  MoveL 5679 to (450.81, 542.83, 100) mm, rotated rx -180 ry 0 rz 160 deg; joints [12.921, 56.747, 9.735, -144.774, 70.43, 166.693]
  Set speed (17.9 mm/s)
  Call Extruder(398.90582)
  MoveL 5680 to (450.02, 541.91, 100) mm, rotated rx 180 ry 0 rz 160 deg; joints [12.82, 56.625, 10.008, -144.909, 70.53, 166.82]
  Set speed (17.9 mm/s)
  Call Extruder(404.31502)
  MoveL 5681 to (448.94, 540.59, 100) mm, rotated rx -180 ry 0 rz 160 deg; joints [12.672, 56.455, 10.386, -145.103, 70.667, 166.997]
  Set speed (17.9 mm/s)
  Call Extruder(407.73007)
  MoveL 5682 to (448.28, 539.73, 100) mm, rotated rx 180 ry 0 rz 160 deg; joints [12.576, 56.35, 10.619, -145.229, 70.751, 167.108]
  Set speed (17.9 mm/s)
  Call Extruder(411.96935)
  MoveL 5683 to (447.47, 538.66, 100) mm, rotated rx -180 ry 0 rz 160 deg; joints [12.453, 56.223, 10.904, -145.387, 70.853, 167.245]
  Set speed (17.9 mm/s)
  Call Extruder(416.06322)
  MoveL 5684 to (446.71, 537.6, 100) mm, rotated rx 180 ry 0 rz 160 deg; joints [12.331, 56.102, 11.173, -145.543, 70.949, 167.375]
  Set speed (17.9 mm/s)
  Call Extruder(420.86880)
  MoveL 5685 to (445.85, 536.35, 100) mm, rotated rx 180 ry 0 rz 160 deg; joints [12.183, 55.965, 11.481, -145.728, 71.057, 167.526]
  Set speed (17.9 mm/s)
  Call Extruder(424.00300)
  MoveL 5686 to (445.3, 535.52, 100) mm, rotated rx 180 ry 0 rz 160 deg; joints [12.084, 55.877, 11.677, -145.851, 71.126, 167.624]
  Set speed (17.9 mm/s)
  Call Extruder(429.28945)
  MoveL 5687 to (444.4, 534.1, 100) mm, rotated rx 180 ry 0 rz 160 deg; joints [11.914, 55.733, 12, -146.061, 71.238, 167.787]
  Set speed (17.9 mm/s)
  Call Extruder(432.98156)
  MoveL 5688 to (443.8, 533.1, 100) mm, rotated rx 180 ry 0 rz 160 deg; joints [11.791, 55.636, 12.219, -146.211, 71.313, 167.899]
  Set speed (17.9 mm/s)
  Call Extruder(437.21112)
  MoveL 5689 to (443.13, 531.94, 100) mm, rotated rx -180 ry 0 rz 160 deg; joints [11.648, 55.527, 12.464, -146.384, 71.396, 168.025]
  Set speed (17.9 mm/s)
  Call Extruder(441.38194)
  MoveL 5690 to (442.49, 530.78, 100) mm, rotated rx -180 ry 0 rz 160 deg; joints [11.504, 55.423, 12.698, -146.557, 71.475, 168.149]
  Set speed (17.9 mm/s)
  Call Extruder(445.63460)
  MoveL 5691 to (441.87, 529.58, 100) mm, rotated rx 180 ry 0 rz 160 deg; joints [11.353, 55.32, 12.93, -146.736, 71.552, 168.273]
  Set speed (17.9 mm/s)
  Call Extruder(449.79410)
  MoveL 5692 to (441.29, 528.4, 100) mm, rotated rx -180 ry 0 rz 160 deg; joints [11.203, 55.223, 13.149, -146.913, 71.624, 168.392]
  Set speed (17.9 mm/s)
  Call Extruder(454.54369)
  MoveL 5693 to (440.65, 527.04, 100) mm, rotated rx -180 ry 0 rz 160 deg; joints [11.028, 55.116, 13.39, -147.118, 71.701, 168.526]
  Set speed (17.9 mm/s)
  Call Extruder(458.16789)
  MoveL 5694 to (440.18, 525.99, 100) mm, rotated rx 180 ry 0 rz 160 deg; joints [10.893, 55.036, 13.571, -147.276, 71.759, 168.627]
  Call Extruder(462.55520)
  MoveL 5695 to (439.64, 524.71, 100) mm, rotated rx -180 ry 0 rz 160 deg; joints [10.725, 54.945, 13.778, -147.469, 71.824, 168.747]
  Call Extruder(466.58097)
  MoveL 5696 to (439.17, 523.52, 100) mm, rotated rx -180 ry 0 rz 160 deg; joints [10.569, 54.863, 13.964, -147.648, 71.881, 168.856]
  Set speed (17.9 mm/s)
  Call Extruder(470.98501)
  MoveL 5697 to (438.69, 522.21, 100) mm, rotated rx -180 ry 0 rz 160 deg; joints [10.395, 54.778, 14.157, -147.847, 71.939, 168.972]
  Set speed (17.9 mm/s)
  Call Extruder(475.05223)
  MoveL 5698 to (438.25, 521, 100) mm, rotated rx -180 ry 0 rz 160 deg; joints [10.233, 54.701, 14.33, -148.031, 71.99, 169.078]
  Set speed (17.9 mm/s)
  Call Extruder(479.39790)
  MoveL 5699 to (437.83, 519.69, 100) mm, rotated rx 180 ry 0 rz 160 deg; joints [10.056, 54.624, 14.505, -148.23, 72.04, 169.189]
  Call Extruder(483.42476)
  MoveL 5700 to (437.45, 518.47, 100) mm, rotated rx 180 ry 0 rz 160 deg; joints [9.891, 54.555, 14.662, -148.416, 72.084, 169.29]
  Set speed (17.9 mm/s)
  Call Extruder(487.83422)
  MoveL 5701 to (437.07, 517.13, 100) mm, rotated rx -180 ry 0 rz 160 deg; joints [9.707, 54.484, 14.823, -148.621, 72.127, 169.398]
  Set speed (17.9 mm/s)
  Call Extruder(491.89983)
  MoveL 5702 to (436.74, 515.89, 100) mm, rotated rx 180 ry 0 rz 160 deg; joints [9.535, 54.421, 14.966, -148.812, 72.164, 169.496]
  Set speed (17.9 mm/s)
  Call Extruder(495.65111)
  MoveL 5703 to (436.47, 514.73, 100) mm, rotated rx -180 ry 0 rz 160 deg; joints [9.375, 54.367, 15.09, -148.989, 72.194, 169.584]
  Set speed (17.8 mm/s)
  Call Extruder(501.06220)
  MoveL 5704 to (436.1, 513.06, 100) mm, rotated rx 180 ry 0 rz 160 deg; joints [9.142, 54.293, 15.259, -149.245, 72.234, 169.709]
  Set speed (17.9 mm/s)
  Call Extruder(508.92492)
  MoveL 5705 to (435.64, 510.61, 100) mm, rotated rx -180 ry 0 rz 160 deg; joints [8.797, 54.196, 15.481, -149.622, 72.28, 169.884]
  Set speed (17.9 mm/s)
  Call Extruder(517.34016)
  MoveL 5706 to (435.26, 507.97, 100) mm, rotated rx 180 ry 0 rz 160 deg; joints [8.421, 54.106, 15.687, -150.03, 72.315, 170.064]
  Set speed (17.9 mm/s)
  Call Extruder(525.75236)
  MoveL 5707 to (435, 505.32, 100) mm, rotated rx 180 ry 0 rz 160 deg; joints [8.039, 54.031, 15.859, -150.44, 72.333, 170.234]
  Set speed (17.9 mm/s)
  Call Extruder(534.00913)
  MoveL 5708 to (434.83, 502.7, 100) mm, rotated rx -180 ry 0 rz 160 deg; joints [7.66, 53.971, 15.996, -150.844, 72.337, 170.393]
  Set speed (17.9 mm/s)
  Call Extruder(542.49356)
  MoveL 5709 to (434.77, 500.01, 100) mm, rotated rx 180 ry 0 rz 160 deg; joints [7.266, 53.923, 16.105, -151.261, 72.325, 170.547]
  Set speed (17.9 mm/s)
  Call Extruder(550.14962)
  MoveL 5710 to (434.82, 497.58, 100) mm, rotated rx 180 ry 0 rz 160 deg; joints [6.909, 53.894, 16.172, -151.637, 72.3, 170.679]
  Set speed (17.9 mm/s)
  Call Extruder(557.57595)
  MoveL 5711 to (434.95, 495.23, 100) mm, rotated rx 180 ry 0 rz 160 deg; joints [6.561, 53.877, 16.21, -152.001, 72.263, 170.799]
  Set speed (17.9 mm/s)
  Call Extruder(565.20370)
  MoveL 5712 to (435.17, 492.83, 100) mm, rotated rx 180 ry 0 rz 160 deg; joints [6.203, 53.871, 16.223, -152.373, 72.213, 170.916]
  Set speed (17.9 mm/s)
  Call Extruder(572.77473)
  MoveL 5713 to (435.48, 490.44, 100) mm, rotated rx -180 ry 0 rz 160 deg; joints [5.847, 53.878, 16.208, -152.741, 72.15, 171.025]
  Call Extruder(580.43460)
  MoveL 5714 to (435.88, 488.05, 100) mm, rotated rx 180 ry 0 rz 160 deg; joints [5.488, 53.897, 16.165, -153.11, 72.072, 171.128]
  Set speed (17.9 mm/s)
  Call Extruder(587.90471)
  MoveL 5715 to (436.36, 485.73, 100) mm, rotated rx -180 ry 0 rz 160 deg; joints [5.139, 53.927, 16.096, -153.466, 71.984, 171.221]
  Set speed (17.9 mm/s)
  Call Extruder(595.43174)
  MoveL 5716 to (436.92, 483.41, 100) mm, rotated rx 180 ry 0 rz 160 deg; joints [4.791, 53.969, 16, -153.821, 71.883, 171.308]
  Set speed (17.9 mm/s)
  Call Extruder(602.95230)
  MoveL 5717 to (437.57, 481.11, 100) mm, rotated rx 180 ry 0 rz 160 deg; joints [4.445, 54.023, 15.877, -154.171, 71.768, 171.389]
  Set speed (17.9 mm/s)
  Call Extruder(610.57330)
  MoveL 5718 to (438.32, 478.81, 100) mm, rotated rx -180 ry 0 rz 160 deg; joints [4.098, 54.089, 15.725, -154.52, 71.64, 171.463]
  Set speed (17.9 mm/s)
  Call Extruder(618.19372)
  MoveL 5719 to (439.14, 476.54, 100) mm, rotated rx -180 ry 0 rz 160 deg; joints [3.756, 54.167, 15.547, -154.862, 71.499, 171.531]
  Set speed (17.9 mm/s)
  Call Extruder(624.98487)
  MoveL 5720 to (439.95, 474.55, 100) mm, rotated rx 180 ry 0 rz 160 deg; joints [3.456, 54.246, 15.366, -155.161, 71.362, 171.585]
  Set speed (17.9 mm/s)
  Call Extruder(633.35469)
  MoveL 5721 to (441.03, 472.13, 100) mm, rotated rx 180 ry 0 rz 160 deg; joints [3.092, 54.357, 15.113, -155.521, 71.18, 171.645]
  Set speed (17.9 mm/s)
  Call Extruder(641.01629)
  MoveL 5722 to (442.11, 469.95, 100) mm, rotated rx 180 ry 0 rz 160 deg; joints [2.766, 54.471, 14.854, -155.842, 71, 171.692]
  Set speed (17.9 mm/s)
  Call Extruder(648.40572)
  MoveL 5723 to (443.23, 467.89, 100) mm, rotated rx -180 ry 0 rz 160 deg; joints [2.458, 54.591, 14.579, -156.142, 70.815, 171.731]
  Call Extruder(655.93186)
  MoveL 5724 to (444.44, 465.84, 100) mm, rotated rx 180 ry 0 rz 160 deg; joints [2.152, 54.725, 14.275, -156.439, 70.615, 171.764]
  Set speed (17.9 mm/s)
  Call Extruder(663.53574)
  MoveL 5725 to (445.74, 463.81, 100) mm, rotated rx -180 ry 0 rz 160 deg; joints [1.85, 54.872, 13.943, -156.73, 70.402, 171.792]
  Set speed (17.9 mm/s)
  Call Extruder(671.21430)
  MoveL 5726 to (447.13, 461.81, 100) mm, rotated rx 180 ry 0 rz 160 deg; joints [1.555, 55.031, 13.583, -157.012, 70.175, 171.813]
  Set speed (17.9 mm/s)
  Call Extruder(678.78294)
  MoveL 5727 to (448.57, 459.89, 100) mm, rotated rx 180 ry 0 rz 160 deg; joints [1.273, 55.199, 13.204, -157.279, 69.94, 171.826]
  Set speed (17.9 mm/s)
  Call Extruder(686.29697)
  MoveL 5728 to (450.07, 458.03, 100) mm, rotated rx 180 ry 0 rz 160 deg; joints [1.003, 55.376, 12.805, -157.533, 69.696, 171.834]
  Set speed (17.9 mm/s)
  Call Extruder(693.99931)
  MoveL 5729 to (451.68, 456.19, 100) mm, rotated rx 180 ry 0 rz 160 deg; joints [0.736, 55.568, 12.372, -157.781, 69.436, 171.835]
  Set speed (17.9 mm/s)
  Call Extruder(701.57500)
  MoveL 5730 to (453.33, 454.44, 100) mm, rotated rx -180 ry 0 rz 160 deg; joints [0.483, 55.767, 11.924, -158.012, 69.17, 171.829]
  Set speed (17.9 mm/s)
  Call Extruder(709.05583)
  MoveL 5731 to (455.02, 452.77, 100) mm, rotated rx -180 ry 0 rz 160 deg; joints [0.245, 55.974, 11.461, -158.228, 68.898, 171.817]
  Set speed (17.9 mm/s)
  Call Extruder(716.62216)
  MoveL 5732 to (456.79, 451.15, 100) mm, rotated rx 180 ry 0 rz 160 deg; joints [0.015, 56.193, 10.971, -158.433, 68.613, 171.798]
  Set speed (17.9 mm/s)
  Call Extruder(724.28486)
  MoveL 5733 to (458.64, 449.58, 100) mm, rotated rx -180 ry 0 rz 160 deg; joints [-0.206, 56.424, 10.454, -158.628, 68.316, 171.773]
  Set speed (17.9 mm/s)
  Call Extruder(731.69796)
  MoveL 5734 to (460.48, 448.12, 100) mm, rotated rx 180 ry 0 rz 160 deg; joints [-0.409, 56.657, 9.935, -158.803, 68.021, 171.741]
  Call Extruder(739.18151)
  MoveL 5735 to (462.39, 446.71, 100) mm, rotated rx -180 ry 0 rz 160 deg; joints [-0.603, 56.901, 9.393, -158.966, 67.715, 171.703]
  Set speed (17.9 mm/s)
  Call Extruder(746.80614)
  MoveL 5736 to (464.4, 445.36, 100) mm, rotated rx 180 ry 0 rz 160 deg; joints [-0.788, 57.159, 8.821, -159.117, 67.395, 171.657]
  Set speed (17.9 mm/s)
  Call Extruder(754.56977)
  MoveL 5737 to (466.48, 444.05, 100) mm, rotated rx -180 ry 0 rz 160 deg; joints [-0.964, 57.431, 8.221, -159.257, 67.062, 171.604]
  Call Extruder(762.12836)
  MoveL 5738 to (468.56, 442.86, 100) mm, rotated rx -180 ry 0 rz 160 deg; joints [-1.122, 57.703, 7.62, -159.378, 66.731, 171.545]
  Set speed (17.9 mm/s)
  Call Extruder(769.52658)
  MoveL 5739 to (470.63, 441.76, 100) mm, rotated rx -180 ry 0 rz 160 deg; joints [-1.266, 57.978, 7.015, -159.483, 66.401, 171.48]
  Call Extruder(777.24414)
  MoveL 5740 to (472.84, 440.7, 100) mm, rotated rx -180 ry 0 rz 160 deg; joints [-1.403, 58.272, 6.369, -159.577, 66.051, 171.405]
  Set speed (17.9 mm/s)
  Call Extruder(784.59819)
  MoveL 5741 to (474.98, 439.77, 100) mm, rotated rx 180 ry 0 rz 160 deg; joints [-1.522, 58.56, 5.738, -159.653, 65.712, 171.327]
  Set speed (17.9 mm/s)
  Call Extruder(792.28153)
  MoveL 5742 to (477.25, 438.88, 100) mm, rotated rx -180 ry 0 rz 160 deg; joints [-1.634, 58.869, 5.065, -159.716, 65.353, 171.238]
  Set speed (17.9 mm/s)
  Call Extruder(800.00638)
  MoveL 5743 to (479.56, 438.07, 100) mm, rotated rx -180 ry 0 rz 160 deg; joints [-1.733, 59.186, 4.374, -159.764, 64.987, 171.141]
  Set speed (17.9 mm/s)
  Call Extruder(807.42236)
  MoveL 5744 to (481.8, 437.37, 100) mm, rotated rx -180 ry 0 rz 160 deg; joints [-1.817, 59.497, 3.698, -159.796, 64.631, 171.04]
  Call Extruder(814.93635)
  MoveL 5745 to (484.1, 436.75, 100) mm, rotated rx 180 ry 0 rz 160 deg; joints [-1.89, 59.818, 3.002, -159.814, 64.268, 170.931]
  Set speed (17.9 mm/s)
  Call Extruder(822.70712)
  MoveL 5746 to (486.5, 436.19, 100) mm, rotated rx -180 ry 0 rz 160 deg; joints [-1.952, 60.156, 2.27, -159.816, 63.889, 170.81]
  Set speed (17.9 mm/s)
  Call Extruder(830.13943)
  MoveL 5747 to (488.82, 435.74, 100) mm, rotated rx 180 ry 0 rz 160 deg; joints [-2, 60.486, 1.559, -159.804, 63.523, 170.687]
  Set speed (17.9 mm/s)
  Call Extruder(837.63896)
  MoveL 5748 to (491.17, 435.38, 100) mm, rotated rx 180 ry 0 rz 160 deg; joints [-2.037, 60.823, 0.833, -159.778, 63.152, 170.555]
  Set speed (17.9 mm/s)
  Call Extruder(845.39030)
  MoveL 5749 to (493.61, 435.09, 100) mm, rotated rx 180 ry 0 rz 160 deg; joints [-2.063, 61.177, 0.074, -159.735, 62.767, 170.41]
  Call Extruder(852.91708)
  MoveL 5750 to (495.99, 434.9, 100) mm, rotated rx 180 ry 0 rz 160 deg; joints [-2.076, 61.525, -0.672, -159.678, 62.392, 170.261]
  Set speed (17.9 mm/s)
  Call Extruder(860.57094)
  MoveL 5751 to (498.41, 434.8, 100) mm, rotated rx 180 ry 0 rz 160 deg; joints [-2.078, 61.883, -1.437, -159.605, 62.01, 170.102]
  Set speed (17.9 mm/s)
  Call Extruder(868.06031)
  MoveL 5752 to (500.79, 434.78, 100) mm, rotated rx 180 ry 0 rz 160 deg; joints [-2.069, 62.237, -2.193, -159.52, 61.636, 169.939]
  Call Extruder(875.70122)
  MoveL 5753 to (503.21, 434.86, 100) mm, rotated rx -180 ry 0 rz 160 deg; joints [-2.049, 62.602, -2.969, -159.419, 61.254, 169.763]
  Set speed (17.9 mm/s)
  Call Extruder(883.20616)
  MoveL 5754 to (505.59, 435.02, 100) mm, rotated rx 180 ry 0 rz 160 deg; joints [-2.018, 62.963, -3.736, -159.305, 60.88, 169.583]
  Set speed (17.9 mm/s)
  Call Extruder(890.83877)
  MoveL 5755 to (508, 435.27, 100) mm, rotated rx 180 ry 0 rz 160 deg; joints [-1.976, 63.333, -4.52, -159.175, 60.501, 169.392]
  Call Extruder(898.35749)
  MoveL 5756 to (510.35, 435.61, 100) mm, rotated rx 180 ry 0 rz 160 deg; joints [-1.924, 63.7, -5.294, -159.033, 60.129, 169.195]
  Set speed (17.9 mm/s)
  Call Extruder(905.98584)
  MoveL 5757 to (512.74, 436.03, 100) mm, rotated rx -180 ry 0 rz 160 deg; joints [-1.861, 64.074, -6.083, -158.876, 59.754, 168.987]
  Call Extruder(913.34804)
  MoveL 5758 to (515.02, 436.53, 100) mm, rotated rx 180 ry 0 rz 160 deg; joints [-1.79, 64.436, -6.845, -158.711, 59.395, 168.779]
  Call Extruder(920.98532)
  MoveL 5759 to (517.37, 437.13, 100) mm, rotated rx 180 ry 0 rz 160 deg; joints [-1.707, 64.813, -7.637, -158.526, 59.025, 168.555]
  Set speed (17.9 mm/s)
  Call Extruder(928.62246)
  MoveL 5760 to (519.69, 437.82, 100) mm, rotated rx 180 ry 0 rz 160 deg; joints [-1.615, 65.19, -8.427, -158.328, 58.659, 168.322]
  Set speed (17.9 mm/s)
  Call Extruder(936.05332)
  MoveL 5761 to (521.92, 438.57, 100) mm, rotated rx -180 ry 0 rz 160 deg; joints [-1.516, 65.557, -9.195, -158.124, 58.307, 168.088]
  Call Extruder(943.74007)
  MoveL 5762 to (524.21, 439.43, 100) mm, rotated rx -180 ry 0 rz 160 deg; joints [-1.404, 65.936, -9.986, -157.899, 57.948, 167.839]
  Set speed (17.9 mm/s)
  Call Extruder(951.26725)
  MoveL 5763 to (526.4, 440.36, 100) mm, rotated rx 180 ry 0 rz 160 deg; joints [-1.286, 66.306, -10.757, -157.667, 57.602, 167.587]
  Call Extruder(958.89094)
  MoveL 5764 to (528.6, 441.38, 100) mm, rotated rx 180 ry 0 rz 160 deg; joints [-1.158, 66.68, -11.534, -157.42, 57.257, 167.324]
  Call Extruder(966.54138)
  MoveL 5765 to (530.76, 442.49, 100) mm, rotated rx -180 ry 0 rz 160 deg; joints [-1.021, 67.053, -12.308, -157.161, 56.917, 167.053]
  Call Extruder(974.10055)
  MoveL 5766 to (532.85, 443.66, 100) mm, rotated rx 180 ry 0 rz 160 deg; joints [-0.878, 67.419, -13.067, -156.894, 56.589, 166.779]
  Set speed (17.9 mm/s)
  Call Extruder(981.59160)
  MoveL 5767 to (534.88, 444.89, 100) mm, rotated rx 180 ry 0 rz 160 deg; joints [-0.728, 67.778, -13.811, -156.618, 56.27, 166.5]
  Set speed (17.9 mm/s)
  Call Extruder(989.24433)
  MoveL 5768 to (536.91, 446.23, 100) mm, rotated rx 180 ry 0 rz 160 deg; joints [-0.567, 68.142, -14.562, -156.326, 55.953, 166.209]
  Set speed (17.9 mm/s)
  Call Extruder(996.72405)
  MoveL 5769 to (538.84, 447.6, 100) mm, rotated rx -180 ry 0 rz 160 deg; joints [-0.404, 68.493, -15.287, -156.032, 55.651, 165.918]
  Set speed (17.9 mm/s)
  Call Extruder(1004.30520)
  MoveL 5770 to (540.75, 449.07, 100) mm, rotated rx -180 ry 0 rz 160 deg; joints [-0.23, 68.845, -16.01, -155.723, 55.354, 165.618]
  Set speed (17.9 mm/s)
  Call Extruder(1011.81497)
  MoveL 5771 to (542.58, 450.59, 100) mm, rotated rx 180 ry 0 rz 160 deg; joints [-0.052, 69.188, -16.715, -155.409, 55.069, 165.316]
  Set speed (17.9 mm/s)
  Call Extruder(1019.44561)
  MoveL 5772 to (544.38, 452.21, 100) mm, rotated rx -180 ry 0 rz 160 deg; joints [0.135, 69.531, -17.419, -155.082, 54.789, 165.005]
  Set speed (17.9 mm/s)
  Call Extruder(1026.97139)
  MoveL 5773 to (546.1, 453.86, 100) mm, rotated rx 180 ry 0 rz 160 deg; joints [0.326, 69.862, -18.098, -154.751, 54.524, 164.693]
  Set speed (17.9 mm/s)
  Call Extruder(1031.19963)
  MoveL 5774 to (547.04, 454.82, 100) mm, rotated rx -180 ry 0 rz 160 deg; joints [0.436, 70.046, -18.474, -154.562, 54.379, 164.516]
  Set speed (17.9 mm/s)
  Call Extruder(1035.37002)
  MoveL 5775 to (547.94, 455.78, 100) mm, rotated rx -180 ry 0 rz 160 deg; joints [0.546, 70.225, -18.84, -154.374, 54.24, 164.341]
  Set speed (17.9 mm/s)
  Call Extruder(1038.63837)
  MoveL 5776 to (548.64, 456.55, 100) mm, rotated rx -180 ry 0 rz 160 deg; joints [0.634, 70.364, -19.124, -154.224, 54.133, 164.202]
  Set speed (17.9 mm/s)
  Call Extruder(1044.28026)
  MoveL 5777 to (549.82, 457.9, 100) mm, rotated rx -180 ry 0 rz 160 deg; joints [0.787, 70.599, -19.605, -153.964, 53.954, 163.962]
  Set speed (17.9 mm/s)
  Call Extruder(1047.97187)
  MoveL 5778 to (550.56, 458.8, 100) mm, rotated rx -180 ry 0 rz 160 deg; joints [0.889, 70.751, -19.915, -153.792, 53.841, 163.805]
  Set speed (17.9 mm/s)
  Call Extruder(1052.40017)
  MoveL 5779 to (551.44, 459.9, 100) mm, rotated rx 180 ry 0 rz 160 deg; joints [1.013, 70.93, -20.281, -153.584, 53.708, 163.615]
  Call Extruder(1056.39533)
  MoveL 5780 to (552.21, 460.91, 100) mm, rotated rx 180 ry 0 rz 160 deg; joints [1.127, 71.089, -20.604, -153.395, 53.593, 163.444]
  Set speed (17.9 mm/s)
  Call Extruder(1060.64284)
  MoveL 5781 to (553, 461.99, 100) mm, rotated rx -180 ry 0 rz 160 deg; joints [1.249, 71.255, -20.943, -153.192, 53.474, 163.261]
  Set speed (17.9 mm/s)
  Call Extruder(1064.81823)
  MoveL 5782 to (553.76, 463.08, 100) mm, rotated rx 180 ry 0 rz 160 deg; joints [1.371, 71.416, -21.269, -152.991, 53.361, 163.081]
  Set speed (17.9 mm/s)
  Call Extruder(1069.00747)
  MoveL 5783 to (554.5, 464.18, 100) mm, rotated rx 180 ry 0 rz 160 deg; joints [1.494, 71.573, -21.59, -152.789, 53.252, 162.9]
  Set speed (17.9 mm/s)
  Call Extruder(1073.69401)
  MoveL 5784 to (555.31, 465.43, 100) mm, rotated rx 180 ry 0 rz 160 deg; joints [1.633, 71.747, -21.942, -152.561, 53.134, 162.698]
  Set speed (17.9 mm/s)
  Call Extruder(1077.43188)
  MoveL 5785 to (555.93, 466.44, 100) mm, rotated rx 180 ry 0 rz 160 deg; joints [1.746, 71.881, -22.216, -152.378, 53.045, 162.537]
  Call Extruder(1081.67784)
  MoveL 5786 to (556.61, 467.6, 100) mm, rotated rx -180 ry 0 rz 160 deg; joints [1.875, 72.031, -22.521, -152.17, 52.947, 162.354]
  Set speed (17.9 mm/s)
  Call Extruder(1087.53287)
  MoveL 5787 to (557.51, 469.23, 100) mm, rotated rx -180 ry 0 rz 160 deg; joints [2.055, 72.233, -22.929, -151.882, 52.819, 162.103]
  Set speed (17.9 mm/s)
  Call Extruder(1090.17409)
  MoveL 5788 to (557.9, 469.97, 100) mm, rotated rx -180 ry 0 rz 160 deg; joints [2.137, 72.321, -23.109, -151.751, 52.764, 161.99]
  Set speed (17.9 mm/s)
  Call Extruder(1094.24936)
  MoveL 5789 to (558.48, 471.12, 100) mm, rotated rx -180 ry 0 rz 160 deg; joints [2.264, 72.454, -23.379, -151.549, 52.683, 161.816]
  Set speed (17.9 mm/s)
  Call Extruder(1098.95352)
  MoveL 5790 to (559.12, 472.47, 100) mm, rotated rx 180 ry 0 rz 160 deg; joints [2.413, 72.604, -23.682, -151.316, 52.595, 161.616]
  Set speed (17.9 mm/s)
  Call Extruder(1102.65916)
  MoveL 5791 to (559.61, 473.54, 100) mm, rotated rx 180 ry 0 rz 160 deg; joints [2.531, 72.718, -23.914, -151.132, 52.529, 161.459]
  Set speed (17.9 mm/s)
  Call Extruder(1107.37343)
  MoveL 5792 to (560.2, 474.91, 100) mm, rotated rx 180 ry 0 rz 160 deg; joints [2.682, 72.858, -24.196, -150.898, 52.452, 161.262]
  Set speed (17.9 mm/s)
  Call Extruder(1111.28917)
  MoveL 5793 to (560.67, 476.06, 100) mm, rotated rx -180 ry 0 rz 160 deg; joints [2.808, 72.972, -24.428, -150.703, 52.391, 161.098]
  Call Extruder(1115.41542)
  MoveL 5794 to (561.13, 477.28, 100) mm, rotated rx 180 ry 0 rz 160 deg; joints [2.943, 73.086, -24.658, -150.499, 52.333, 160.928]
  Set speed (17.9 mm/s)
  Call Extruder(1119.53817)
  MoveL 5795 to (561.58, 478.5, 100) mm, rotated rx -180 ry 0 rz 160 deg; joints [3.077, 73.199, -24.885, -150.294, 52.278, 160.758]
  Set speed (17.9 mm/s)
  Call Extruder(1123.83675)
  MoveL 5796 to (562.01, 479.8, 100) mm, rotated rx -180 ry 0 rz 160 deg; joints [3.219, 73.308, -25.107, -150.082, 52.227, 160.584]
  Call Extruder(1128.03874)
  MoveL 5797 to (562.41, 481.06, 100) mm, rotated rx 180 ry 0 rz 160 deg; joints [3.358, 73.414, -25.32, -149.875, 52.18, 160.414]
  Set speed (17.9 mm/s)
  Call Extruder(1132.22902)
  MoveL 5798 to (562.78, 482.34, 100) mm, rotated rx -180 ry 0 rz 160 deg; joints [3.497, 73.512, -25.518, -149.669, 52.141, 160.248]
  Set speed (17.9 mm/s)
  Call Extruder(1136.26465)
  MoveL 5799 to (563.12, 483.57, 100) mm, rotated rx 180 ry 0 rz 160 deg; joints [3.632, 73.605, -25.705, -149.471, 52.106, 160.089]
  Call Extruder(1140.67454)
  MoveL 5800 to (563.45, 484.93, 100) mm, rotated rx -180 ry 0 rz 160 deg; joints [3.781, 73.698, -25.895, -149.256, 52.074, 159.918]
  Call Extruder(1144.77390)
  MoveL 5801 to (563.74, 486.19, 100) mm, rotated rx 180 ry 0 rz 160 deg; joints [3.919, 73.784, -26.066, -149.057, 52.048, 159.761]
  Set speed (17.9 mm/s)
  Call Extruder(1153.44625)
  MoveL 5802 to (564.27, 488.89, 100) mm, rotated rx 180 ry 0 rz 160 deg; joints [4.215, 73.945, -26.391, -148.639, 52.01, 159.437]
  Set speed (17.9 mm/s)
  Call Extruder(1161.67703)
  MoveL 5803 to (564.66, 491.47, 100) mm, rotated rx 180 ry 0 rz 160 deg; joints [4.498, 74.078, -26.66, -148.248, 51.995, 159.14]
  Call Extruder(1170.18168)
  MoveL 5804 to (564.96, 494.15, 100) mm, rotated rx -180 ry 0 rz 160 deg; joints [4.792, 74.196, -26.897, -147.85, 51.999, 158.845]
  Call Extruder(1178.50578)
  MoveL 5805 to (565.14, 496.79, 100) mm, rotated rx 180 ry 0 rz 160 deg; joints [5.082, 74.29, -27.086, -147.468, 52.024, 158.57]
  Set speed (17.9 mm/s)
  Call Extruder(1186.85602)
  MoveL 5806 to (565.22, 499.43, 100) mm, rotated rx 180 ry 0 rz 160 deg; joints [5.373, 74.362, -27.232, -147.093, 52.069, 158.308]
  Set speed (17.9 mm/s)
  Call Extruder(1195.19846)
  MoveL 5807 to (565.19, 502.08, 100) mm, rotated rx -180 ry 0 rz 160 deg; joints [5.665, 74.414, -27.336, -146.727, 52.134, 158.061]
  Set speed (17.9 mm/s)
  Call Extruder(1203.73141)
  MoveL 5808 to (565.05, 504.78, 100) mm, rotated rx 180 ry 0 rz 160 deg; joints [5.965, 74.445, -27.399, -146.362, 52.22, 157.824]
  Set speed (17.9 mm/s)
  Call Extruder(1212.05652)
  MoveL 5809 to (564.8, 507.41, 100) mm, rotated rx -180 ry 0 rz 160 deg; joints [6.258, 74.453, -27.414, -146.016, 52.325, 157.609]
  Set speed (17.9 mm/s)
  Call Extruder(1220.63729)
  MoveL 5810 to (564.43, 510.11, 100) mm, rotated rx -180 ry 0 rz 160 deg; joints [6.559, 74.438, -27.385, -145.671, 52.453, 157.404]
  Call Extruder(1229.19039)
  MoveL 5811 to (563.96, 512.78, 100) mm, rotated rx 180 ry 0 rz 160 deg; joints [6.859, 74.401, -27.31, -145.338, 52.599, 157.219]
  Call Extruder(1237.40699)
  MoveL 5812 to (563.39, 515.33, 100) mm, rotated rx 180 ry 0 rz 160 deg; joints [7.147, 74.344, -27.195, -145.03, 52.759, 157.058]
  Set speed (17.9 mm/s)
  Call Extruder(1245.34913)
  MoveL 5813 to (562.76, 517.76, 100) mm, rotated rx -180 ry 0 rz 160 deg; joints [7.424, 74.269, -27.045, -144.743, 52.928, 156.92]
  Set speed (17.9 mm/s)
  Call Extruder(1250.95485)
  MoveL 5814 to (562.25, 519.46, 100) mm, rotated rx 180 ry 0 rz 160 deg; joints [7.618, 74.204, -26.914, -144.548, 53.059, 156.833]
  Set speed (17.9 mm/s)
  Call Extruder(1254.21125)
  MoveL 5815 to (561.94, 520.45, 100) mm, rotated rx 180 ry 0 rz 160 deg; joints [7.731, 74.164, -26.833, -144.436, 53.136, 156.785]
  Call Extruder(1258.88399)
  MoveL 5816 to (561.45, 521.84, 100) mm, rotated rx 180 ry 0 rz 160 deg; joints [7.892, 74.097, -26.698, -144.281, 53.255, 156.723]
  Set speed (17.9 mm/s)
  Call Extruder(1262.79210)
  MoveL 5817 to (561.03, 523.01, 100) mm, rotated rx -180 ry 0 rz 160 deg; joints [8.027, 74.039, -26.581, -144.152, 53.356, 156.674]
  Set speed (17.9 mm/s)
  Call Extruder(1267.25552)
  MoveL 5818 to (560.51, 524.33, 100) mm, rotated rx 180 ry 0 rz 160 deg; joints [8.18, 73.965, -26.431, -144.01, 53.478, 156.625]
  Call Extruder(1270.87292)
  MoveL 5819 to (560.08, 525.39, 100) mm, rotated rx 180 ry 0 rz 160 deg; joints [8.304, 73.902, -26.306, -143.896, 53.578, 156.587]
  Call Extruder(1275.66647)
  MoveL 5820 to (559.47, 526.78, 100) mm, rotated rx 180 ry 0 rz 160 deg; joints [8.467, 73.812, -26.123, -143.75, 53.718, 156.544]
  Set speed (17.9 mm/s)
  Call Extruder(1279.88602)
  MoveL 5821 to (558.91, 527.99, 100) mm, rotated rx -180 ry 0 rz 160 deg; joints [8.61, 73.729, -25.955, -143.624, 53.843, 156.51]
  Set speed (17.9 mm/s)
  Call Extruder(1283.61536)
  MoveL 5822 to (558.39, 529.06, 100) mm, rotated rx -180 ry 0 rz 160 deg; joints [8.736, 73.65, -25.796, -143.516, 53.957, 156.485]
  Set speed (17.9 mm/s)
  Call Extruder(1287.99352)
  MoveL 5823 to (557.76, 530.29, 100) mm, rotated rx -180 ry 0 rz 160 deg; joints [8.884, 73.552, -25.6, -143.392, 54.096, 156.46]
  Set speed (17.9 mm/s)
  Call Extruder(1292.53711)
  MoveL 5824 to (557.07, 531.56, 100) mm, rotated rx 180 ry 0 rz 160 deg; joints [9.035, 73.446, -25.385, -143.267, 54.244, 156.439]
  Call Extruder(1296.24969)
  MoveL 5825 to (556.5, 532.59, 100) mm, rotated rx -180 ry 0 rz 160 deg; joints [9.159, 73.355, -25.202, -143.167, 54.367, 156.426]
  Set speed (17.9 mm/s)
  Call Extruder(1300.41758)
  MoveL 5826 to (555.83, 533.73, 100) mm, rotated rx -180 ry 0 rz 160 deg; joints [9.297, 73.25, -24.988, -143.058, 54.508, 156.415]
  Set speed (17.9 mm/s)
  Call Extruder(1304.83583)
  MoveL 5827 to (555.09, 534.92, 100) mm, rotated rx -180 ry 0 rz 160 deg; joints [9.442, 73.133, -24.752, -142.946, 54.662, 156.409]
  Set speed (17.9 mm/s)
  Call Extruder(1308.83293)
  MoveL 5828 to (554.4, 535.99, 100) mm, rotated rx -180 ry 0 rz 160 deg; joints [9.572, 73.022, -24.529, -142.848, 54.804, 156.407]
  Set speed (17.9 mm/s)
  Call Extruder(1313.12375)
  MoveL 5829 to (553.63, 537.11, 100) mm, rotated rx 180 ry 0 rz 160 deg; joints [9.711, 72.899, -24.28, -142.746, 54.96, 156.411]
  Set speed (17.9 mm/s)
  Call Extruder(1317.41236)
  MoveL 5830 to (552.85, 538.22, 100) mm, rotated rx 180 ry 0 rz 160 deg; joints [9.849, 72.773, -24.024, -142.646, 55.118, 156.418]
  Set speed (17.9 mm/s)
  Call Extruder(1322.92340)
  MoveL 5831 to (551.81, 539.63, 100) mm, rotated rx 180 ry 0 rz 160 deg; joints [10.025, 72.604, -23.682, -142.523, 55.326, 156.434]
  Set speed (17.9 mm/s)
  Call Extruder(1325.83347)
  MoveL 5832 to (551.24, 540.35, 100) mm, rotated rx 180 ry 0 rz 160 deg; joints [10.117, 72.512, -23.496, -142.461, 55.437, 156.446]
  Set speed (17.9 mm/s)
  Call Extruder(1329.94289)
  MoveL 5833 to (550.43, 541.37, 100) mm, rotated rx -180 ry 0 rz 160 deg; joints [10.246, 72.379, -23.226, -142.375, 55.597, 156.466]
  Set speed (17.9 mm/s)
  Call Extruder(1335.20101)
  MoveL 5834 to (549.35, 542.65, 100) mm, rotated rx -180 ry 0 rz 160 deg; joints [10.41, 72.204, -22.871, -142.268, 55.805, 156.497]
  Set speed (17.9 mm/s)
  Call Extruder(1338.74944)
  MoveL 5835 to (548.61, 543.49, 100) mm, rotated rx 180 ry 0 rz 160 deg; joints [10.519, 72.082, -22.623, -142.199, 55.948, 156.522]
  Set speed (17.9 mm/s)
  Call Extruder(1342.97071)
  MoveL 5836 to (547.7, 544.48, 100) mm, rotated rx 180 ry 0 rz 160 deg; joints [10.648, 71.933, -22.322, -142.12, 56.12, 156.556]
  Set speed (17.9 mm/s)
  Call Extruder(1347.16725)
  MoveL 5837 to (546.79, 545.44, 100) mm, rotated rx -180 ry 0 rz 160 deg; joints [10.774, 71.783, -22.017, -142.044, 56.292, 156.592]
  Set speed (17.9 mm/s)
  Call Extruder(1350.92435)
  MoveL 5838 to (545.95, 546.29, 100) mm, rotated rx 180 ry 0 rz 160 deg; joints [10.887, 71.645, -21.737, -141.978, 56.449, 156.629]
  Set speed (17.9 mm/s)
  Call Extruder(1355.12158)
  MoveL 5839 to (545, 547.22, 100) mm, rotated rx -180 ry 0 rz 160 deg; joints [11.011, 71.489, -21.418, -141.907, 56.626, 156.673]
  Set speed (17.9 mm/s)
  Call Extruder(1359.46484)
  MoveL 5840 to (543.99, 548.16, 100) mm, rotated rx -180 ry 0 rz 160 deg; joints [11.138, 71.323, -21.08, -141.837, 56.811, 156.724]
  Set speed (17.9 mm/s)
  Call Extruder(1363.56091)
  MoveL 5841 to (543.02, 549.02, 100) mm, rotated rx -180 ry 0 rz 160 deg; joints [11.256, 71.164, -20.756, -141.774, 56.988, 156.774]
  Call Extruder(1367.80541)
  MoveL 5842 to (542, 549.9, 100) mm, rotated rx 180 ry 0 rz 160 deg; joints [11.377, 70.996, -20.415, -141.711, 57.172, 156.83]
  Set speed (17.9 mm/s)
  Call Extruder(1371.93527)
  MoveL 5843 to (540.99, 550.73, 100) mm, rotated rx 180 ry 0 rz 160 deg; joints [11.494, 70.83, -20.076, -141.653, 57.353, 156.889]
  Call Extruder(1376.11842)
  MoveL 5844 to (539.95, 551.56, 100) mm, rotated rx -180 ry 0 rz 160 deg; joints [11.61, 70.659, -19.728, -141.596, 57.538, 156.951]
  Set speed (17.9 mm/s)
  Call Extruder(1380.34094)
  MoveL 5845 to (538.88, 552.37, 100) mm, rotated rx 180 ry 0 rz 160 deg; joints [11.726, 70.484, -19.371, -141.541, 57.726, 157.018]
  Call Extruder(1384.78388)
  MoveL 5846 to (537.74, 553.2, 100) mm, rotated rx -180 ry 0 rz 160 deg; joints [11.846, 70.298, -18.989, -141.487, 57.925, 157.092]
  Set speed (17.9 mm/s)
  Call Extruder(1389.23338)
  MoveL 5847 to (536.58, 554, 100) mm, rotated rx 180 ry 0 rz 160 deg; joints [11.964, 70.108, -18.6, -141.436, 58.127, 157.17]
  Set speed (17.9 mm/s)
  Call Extruder(1392.85535)
  MoveL 5848 to (535.62, 554.64, 100) mm, rotated rx -180 ry 0 rz 160 deg; joints [12.059, 69.951, -18.281, -141.396, 58.291, 157.235]
  Set speed (17.9 mm/s)
  Call Extruder(1397.17836)
  MoveL 5849 to (534.47, 555.37, 100) mm, rotated rx 180 ry 0 rz 160 deg; joints [12.17, 69.763, -17.894, -141.352, 58.489, 157.317]
  Set speed (17.9 mm/s)
  Call Extruder(1401.83512)
  MoveL 5850 to (533.21, 556.14, 100) mm, rotated rx 180 ry 0 rz 160 deg; joints [12.288, 69.557, -17.473, -141.307, 58.702, 157.409]
  Set speed (17.9 mm/s)
  Call Extruder(1405.59771)
  MoveL 5851 to (532.17, 556.74, 100) mm, rotated rx -180 ry 0 rz 160 deg; joints [12.382, 69.389, -17.127, -141.273, 58.876, 157.486]
  Set speed (17.9 mm/s)
  Call Extruder(1409.23758)
  MoveL 5852 to (531.16, 557.3, 100) mm, rotated rx 180 ry 0 rz 160 deg; joints [12.471, 69.225, -16.791, -141.242, 59.045, 157.562]
  Set speed (17.9 mm/s)
  Call Extruder(1414.04469)
  MoveL 5853 to (529.82, 558.01, 100) mm, rotated rx 180 ry 0 rz 160 deg; joints [12.586, 69.006, -16.342, -141.204, 59.269, 157.667]
  Call Extruder(1418.67857)
  MoveL 5854 to (528.5, 558.66, 100) mm, rotated rx -180 ry 0 rz 160 deg; joints [12.694, 68.793, -15.904, -141.171, 59.485, 157.772]
  Set speed (17.9 mm/s)
  Call Extruder(1422.53414)
  MoveL 5855 to (527.4, 559.19, 100) mm, rotated rx 180 ry 0 rz 160 deg; joints [12.783, 68.615, -15.536, -141.146, 59.666, 157.861]
  Set speed (17.9 mm/s)
  Call Extruder(1426.70274)
  MoveL 5856 to (526.19, 559.73, 100) mm, rotated rx -180 ry 0 rz 160 deg; joints [12.876, 68.42, -15.135, -141.122, 59.861, 157.961]
  Set speed (17.9 mm/s)
  Call Extruder(1430.81868)
  MoveL 5857 to (524.99, 560.24, 100) mm, rotated rx -180 ry 0 rz 160 deg; joints [12.966, 68.227, -14.738, -141.099, 60.054, 158.06]
  Set speed (17.9 mm/s)
  Call Extruder(1435.12111)
  MoveL 5858 to (523.73, 560.75, 100) mm, rotated rx 180 ry 0 rz 160 deg; joints [13.058, 68.024, -14.318, -141.079, 60.257, 158.168]
  Set speed (17.9 mm/s)
  Call Extruder(1439.34950)
  MoveL 5859 to (522.48, 561.23, 100) mm, rotated rx -180 ry 0 rz 160 deg; joints [13.146, 67.823, -13.904, -141.06, 60.456, 158.276]
  Set speed (17.9 mm/s)
  Call Extruder(1443.96614)
  MoveL 5860 to (521.1, 561.71, 100) mm, rotated rx 180 ry 0 rz 160 deg; joints [13.239, 67.602, -13.447, -141.045, 60.674, 158.398]
  Call Extruder(1447.75239)
  MoveL 5861 to (519.96, 562.09, 100) mm, rotated rx 180 ry 0 rz 160 deg; joints [13.315, 67.421, -13.072, -141.033, 60.852, 158.498]
  Set speed (17.9 mm/s)
  Call Extruder(1456.11391)
  MoveL 5862 to (517.42, 562.85, 100) mm, rotated rx -180 ry 0 rz 160 deg; joints [13.473, 67.016, -12.233, -141.016, 61.247, 158.729]
  Set speed (17.9 mm/s)
  Call Extruder(1459.84226)
  MoveL 5863 to (516.28, 563.15, 100) mm, rotated rx 180 ry 0 rz 160 deg; joints [13.539, 66.834, -11.856, -141.012, 61.423, 158.835]
  Set speed (17.9 mm/s)
  Call Extruder(1464.46214)
  MoveL 5864 to (514.86, 563.51, 100) mm, rotated rx -180 ry 0 rz 160 deg; joints [13.62, 66.61, -11.389, -141.009, 61.641, 158.967]
  Set speed (17.9 mm/s)
  Call Extruder(1473.02091)
  MoveL 5865 to (512.21, 564.07, 100) mm, rotated rx -180 ry 0 rz 160 deg; joints [13.762, 66.19, -10.516, -141.012, 62.044, 159.22]
  Call Extruder(1481.48428)
  MoveL 5866 to (509.56, 564.52, 100) mm, rotated rx 180 ry 0 rz 160 deg; joints [13.891, 65.774, -9.647, -141.025, 62.441, 159.478]
  Call Extruder(1489.72627)
  MoveL 5867 to (506.97, 564.85, 100) mm, rotated rx 180 ry 0 rz 160 deg; joints [14.006, 65.367, -8.797, -141.048, 62.825, 159.736]
  Set speed (17.9 mm/s)
  Call Extruder(1498.27519)
  MoveL 5868 to (504.26, 565.08, 100) mm, rotated rx -180 ry 0 rz 160 deg; joints [14.114, 64.945, -7.913, -141.082, 63.222, 160.01]
  Call Extruder(1506.73394)
  MoveL 5869 to (501.58, 565.2, 100) mm, rotated rx 180 ry 0 rz 160 deg; joints [14.209, 64.527, -7.037, -141.126, 63.611, 160.287]
  Set speed (17.9 mm/s)
  Call Extruder(1514.95462)
  MoveL 5870 to (498.98, 565.21, 100) mm, rotated rx 180 ry 0 rz 160 deg; joints [14.289, 64.123, -6.186, -141.179, 63.986, 160.562]
  Set speed (10.0 mm/s)
  MoveL 5871 to (498.98, 565.21, 104) mm, rotated rx 180 ry 0 rz 160 deg; joints [14.289, 63.491, -5.899, -141.073, 63.717, 160.321]
  Set speed (120.0 mm/s)
  MoveL 5872 to (498.98, 564.59, 104) mm, rotated rx -180 ry 0 rz 160 deg; joints [14.214, 63.467, -5.849, -141.16, 63.712, 160.374]
  Set speed (17.6 mm/s)
  Call Extruder(1523.55152)
  MoveL 5873 to (496.3, 564.49, 104) mm, rotated rx 180 ry 0 rz 160 deg; joints [14.285, 63.05, -4.975, -141.226, 64.092, 160.66]
  Set speed (17.6 mm/s)
  Call Extruder(1532.03521)
  MoveL 5874 to (493.65, 564.29, 104) mm, rotated rx 180 ry 0 rz 160 deg; joints [14.341, 62.641, -4.116, -141.302, 64.462, 160.947]
  Call Extruder(1540.42814)
  MoveL 5875 to (491.05, 563.98, 104) mm, rotated rx 180 ry 0 rz 160 deg; joints [14.385, 62.239, -3.269, -141.389, 64.823, 161.235]
  Set speed (17.6 mm/s)
  Call Extruder(1548.78688)
  MoveL 5876 to (488.47, 563.56, 104) mm, rotated rx 180 ry 0 rz 160 deg; joints [14.415, 61.841, -2.43, -141.486, 65.178, 161.525]
  Set speed (17.6 mm/s)
  Call Extruder(1557.21308)
  MoveL 5877 to (485.89, 563.04, 104) mm, rotated rx 180 ry 0 rz 160 deg; joints [14.432, 61.444, -1.59, -141.594, 65.53, 161.821]
  Set speed (17.6 mm/s)
  Call Extruder(1561.62651)
  MoveL 5878 to (484.55, 562.72, 104) mm, rotated rx -180 ry 0 rz 160 deg; joints [14.435, 61.238, -1.153, -141.655, 65.712, 161.977]
  Set speed (17.6 mm/s)
  Call Extruder(1565.84704)
  MoveL 5879 to (483.27, 562.4, 104) mm, rotated rx 180 ry 0 rz 160 deg; joints [14.436, 61.042, -0.738, -141.716, 65.884, 162.126]
  Set speed (17.6 mm/s)
  Call Extruder(1574.11726)
  MoveL 5880 to (480.8, 561.68, 104) mm, rotated rx 180 ry 0 rz 160 deg; joints [14.426, 60.661, 0.071, -141.844, 66.218, 162.42]
  Call Extruder(0.00000)
  Set speed (17.6 mm/s)
  Call Extruder(4.38070)
  MoveL 5881 to (479.5, 561.25, 104) mm, rotated rx -180 ry 0 rz 160 deg; joints [14.414, 60.462, 0.496, -141.917, 66.391, 162.577]
  Call Extruder(8.59213)
  MoveL 5882 to (478.25, 560.83, 104) mm, rotated rx -180 ry 0 rz 160 deg; joints [14.402, 60.271, 0.901, -141.988, 66.557, 162.727]
  Set speed (17.6 mm/s)
  Call Extruder(12.89777)
  MoveL 5883 to (477, 560.36, 104) mm, rotated rx 180 ry 0 rz 160 deg; joints [14.383, 60.078, 1.313, -142.066, 66.724, 162.881]
  Call Extruder(17.56272)
  MoveL 5884 to (475.64, 559.83, 104) mm, rotated rx 180 ry 0 rz 160 deg; joints [14.36, 59.871, 1.757, -142.151, 66.904, 163.048]
  Set speed (17.6 mm/s)
  Call Extruder(24.42718)
  MoveL 5885 to (473.67, 558.99, 104) mm, rotated rx -180 ry 0 rz 160 deg; joints [14.318, 59.569, 2.403, -142.285, 67.163, 163.294]
  Set speed (17.6 mm/s)
  Call Extruder(29.78772)
  MoveL 5886 to (472.15, 558.29, 104) mm, rotated rx -180 ry 0 rz 160 deg; joints [14.277, 59.337, 2.902, -142.395, 67.363, 163.487]
  Set speed (17.6 mm/s)
  Call Extruder(34.03995)
  MoveL 5887 to (470.96, 557.7, 104) mm, rotated rx 180 ry 0 rz 160 deg; joints [14.241, 59.154, 3.294, -142.486, 67.518, 163.64]
  Set speed (17.6 mm/s)
  Call Extruder(37.07804)
  MoveL 5888 to (470.11, 557.27, 104) mm, rotated rx -180 ry 0 rz 160 deg; joints [14.213, 59.025, 3.572, -142.552, 67.629, 163.749]
  Set speed (17.6 mm/s)
  Call Extruder(42.46990)
  MoveL 5889 to (468.63, 556.47, 104) mm, rotated rx 180 ry 0 rz 160 deg; joints [14.158, 58.798, 4.061, -142.675, 67.821, 163.942]
  Set speed (17.6 mm/s)
  Call Extruder(46.64346)
  MoveL 5890 to (467.5, 555.83, 104) mm, rotated rx 180 ry 0 rz 160 deg; joints [14.112, 58.624, 4.436, -142.772, 67.969, 164.091]
  Set speed (17.6 mm/s)
  Call Extruder(50.97222)
  MoveL 5891 to (466.34, 555.13, 104) mm, rotated rx 180 ry 0 rz 160 deg; joints [14.06, 58.445, 4.82, -142.876, 68.119, 164.246]
  Call Extruder(55.12272)
  MoveL 5892 to (465.23, 554.44, 104) mm, rotated rx -180 ry 0 rz 160 deg; joints [14.007, 58.277, 5.185, -142.979, 68.261, 164.394]
  Set speed (17.6 mm/s)
  Call Extruder(59.28151)
  MoveL 5893 to (464.15, 553.73, 104) mm, rotated rx 180 ry 0 rz 160 deg; joints [13.949, 58.109, 5.547, -143.085, 68.401, 164.542]
  Set speed (17.6 mm/s)
  Call Extruder(63.60438)
  MoveL 5894 to (463.03, 552.97, 104) mm, rotated rx 180 ry 0 rz 160 deg; joints [13.886, 57.938, 5.919, -143.198, 68.544, 164.695]
  Set speed (17.6 mm/s)
  Call Extruder(67.83859)
  MoveL 5895 to (461.95, 552.2, 104) mm, rotated rx 180 ry 0 rz 160 deg; joints [13.82, 57.772, 6.278, -143.311, 68.682, 164.844]
  Set speed (17.6 mm/s)
  Call Extruder(72.06876)
  MoveL 5896 to (460.89, 551.41, 104) mm, rotated rx 180 ry 0 rz 160 deg; joints [13.75, 57.609, 6.633, -143.428, 68.818, 164.993]
  Set speed (17.6 mm/s)
  Call Extruder(76.24508)
  MoveL 5897 to (459.86, 550.62, 104) mm, rotated rx -180 ry 0 rz 160 deg; joints [13.678, 57.45, 6.979, -143.546, 68.949, 165.139]
  Set speed (17.6 mm/s)
  Call Extruder(80.42942)
  MoveL 5898 to (458.85, 549.79, 104) mm, rotated rx -180 ry 0 rz 160 deg; joints [13.602, 57.293, 7.321, -143.667, 69.079, 165.285]
  Set speed (17.6 mm/s)
  Call Extruder(84.74088)
  MoveL 5899 to (457.82, 548.92, 104) mm, rotated rx -180 ry 0 rz 160 deg; joints [13.519, 57.133, 7.668, -143.795, 69.209, 165.435]
  Set speed (17.6 mm/s)
  Call Extruder(89.01165)
  MoveL 5900 to (456.82, 548.04, 104) mm, rotated rx -180 ry 0 rz 160 deg; joints [13.434, 56.978, 8.007, -143.924, 69.337, 165.582]
  Call Extruder(93.17335)
  MoveL 5901 to (455.86, 547.16, 104) mm, rotated rx 180 ry 0 rz 160 deg; joints [13.347, 56.829, 8.333, -144.054, 69.458, 165.724]
  Set speed (17.6 mm/s)
  Call Extruder(97.79900)
  MoveL 5902 to (454.81, 546.16, 104) mm, rotated rx 180 ry 0 rz 160 deg; joints [13.246, 56.667, 8.688, -144.2, 69.589, 165.882]
  Call Extruder(102.76295)
  MoveL 5903 to (453.72, 545.06, 104) mm, rotated rx 180 ry 0 rz 160 deg; joints [13.132, 56.495, 9.063, -144.361, 69.728, 166.049]
  Call Extruder(105.91320)
  MoveL 5904 to (453.04, 544.35, 104) mm, rotated rx -180 ry 0 rz 160 deg; joints [13.058, 56.389, 9.297, -144.466, 69.813, 166.155]
  Set speed (17.6 mm/s)
  Call Extruder(110.12997)
  MoveL 5905 to (452.14, 543.39, 104) mm, rotated rx 180 ry 0 rz 160 deg; joints [12.955, 56.249, 9.605, -144.608, 69.925, 166.295]
  Call Extruder(114.40516)
  MoveL 5906 to (451.25, 542.39, 104) mm, rotated rx -180 ry 0 rz 160 deg; joints [12.847, 56.109, 9.912, -144.755, 70.036, 166.437]
  Call Extruder(118.54807)
  MoveL 5907 to (450.41, 541.4, 104) mm, rotated rx 180 ry 0 rz 160 deg; joints [12.739, 55.977, 10.204, -144.9, 70.141, 166.572]
  Set speed (17.6 mm/s)
  Call Extruder(122.84948)
  MoveL 5908 to (449.56, 540.36, 104) mm, rotated rx 180 ry 0 rz 160 deg; joints [12.623, 55.842, 10.501, -145.054, 70.247, 166.712]
  Set speed (17.6 mm/s)
  Call Extruder(127.03277)
  MoveL 5909 to (448.76, 539.33, 104) mm, rotated rx -180 ry 0 rz 160 deg; joints [12.506, 55.714, 10.783, -145.206, 70.347, 166.846]
  Set speed (17.6 mm/s)
  Call Extruder(131.22892)
  MoveL 5910 to (447.97, 538.29, 104) mm, rotated rx 180 ry 0 rz 160 deg; joints [12.386, 55.588, 11.061, -145.361, 70.445, 166.98]
  Set speed (17.6 mm/s)
  Call Extruder(135.84203)
  MoveL 5911 to (447.13, 537.12, 104) mm, rotated rx 180 ry 0 rz 160 deg; joints [12.25, 55.454, 11.359, -145.534, 70.549, 167.125]
  Set speed (17.6 mm/s)
  Call Extruder(140.75155)
  MoveL 5912 to (446.26, 535.85, 104) mm, rotated rx 180 ry 0 rz 160 deg; joints [12.101, 55.314, 11.668, -145.722, 70.656, 167.278]
  Call Extruder(144.34775)
  MoveL 5913 to (445.65, 534.91, 104) mm, rotated rx 180 ry 0 rz 160 deg; joints [11.989, 55.215, 11.888, -145.862, 70.732, 167.388]
  Set speed (17.6 mm/s)
  Call Extruder(148.51476)
  MoveL 5914 to (444.95, 533.8, 104) mm, rotated rx -180 ry 0 rz 160 deg; joints [11.856, 55.102, 12.139, -146.026, 70.817, 167.515]
  Call Extruder(152.45745)
  MoveL 5915 to (444.32, 532.75, 104) mm, rotated rx -180 ry 0 rz 160 deg; joints [11.727, 54.998, 12.369, -146.184, 70.894, 167.633]
  Set speed (17.6 mm/s)
  Call Extruder(156.04014)
  MoveL 5916 to (443.76, 531.78, 104) mm, rotated rx -180 ry 0 rz 160 deg; joints [11.608, 54.906, 12.574, -146.329, 70.962, 167.74]
  Set speed (17.6 mm/s)
  Call Extruder(160.78233)
  MoveL 5917 to (443.04, 530.48, 104) mm, rotated rx -180 ry 0 rz 160 deg; joints [11.447, 54.788, 12.837, -146.523, 71.049, 167.879]
  Set speed (17.6 mm/s)
  Call Extruder(165.08763)
  MoveL 5918 to (442.43, 529.29, 104) mm, rotated rx -180 ry 0 rz 160 deg; joints [11.297, 54.684, 13.068, -146.702, 71.124, 168.003]
  Set speed (17.6 mm/s)
  Call Extruder(169.38215)
  MoveL 5919 to (441.83, 528.09, 104) mm, rotated rx -180 ry 0 rz 160 deg; joints [11.144, 54.584, 13.291, -146.883, 71.196, 168.126]
  Set speed (17.6 mm/s)
  Call Extruder(173.61397)
  MoveL 5920 to (441.27, 526.89, 104) mm, rotated rx 180 ry 0 rz 160 deg; joints [10.99, 54.489, 13.503, -147.063, 71.262, 168.244]
  Set speed (17.6 mm/s)
  Call Extruder(177.84959)
  MoveL 5921 to (440.73, 525.69, 104) mm, rotated rx 180 ry 0 rz 160 deg; joints [10.835, 54.397, 13.71, -147.245, 71.327, 168.361]
  Set speed (17.6 mm/s)
  Call Extruder(182.08554)
  MoveL 5922 to (440.22, 524.47, 104) mm, rotated rx -180 ry 0 rz 160 deg; joints [10.675, 54.309, 13.908, -147.43, 71.387, 168.476]
  Set speed (17.6 mm/s)
  Call Extruder(186.12743)
  MoveL 5923 to (439.75, 523.3, 104) mm, rotated rx -180 ry 0 rz 160 deg; joints [10.521, 54.227, 14.091, -147.607, 71.442, 168.584]
  Set speed (17.6 mm/s)
  Call Extruder(190.55205)
  MoveL 5924 to (439.27, 522, 104) mm, rotated rx -180 ry 0 rz 160 deg; joints [10.349, 54.142, 14.282, -147.804, 71.497, 168.7]
  Call Extruder(194.64698)
  MoveL 5925 to (438.84, 520.8, 104) mm, rotated rx 180 ry 0 rz 160 deg; joints [10.189, 54.065, 14.454, -147.987, 71.547, 168.806]
  Set speed (17.6 mm/s)
  Call Extruder(199.01037)
  MoveL 5926 to (438.42, 519.5, 104) mm, rotated rx 180 ry 0 rz 160 deg; joints [10.014, 53.988, 14.627, -148.185, 71.594, 168.917]
  Set speed (17.6 mm/s)
  Call Extruder(203.11258)
  MoveL 5927 to (438.04, 518.28, 104) mm, rotated rx 180 ry 0 rz 160 deg; joints [9.849, 53.917, 14.785, -148.371, 71.637, 169.02]
  Set speed (17.6 mm/s)
  Call Extruder(207.49396)
  MoveL 5928 to (437.68, 516.97, 104) mm, rotated rx 180 ry 0 rz 160 deg; joints [9.668, 53.848, 14.942, -148.573, 71.677, 169.126]
  Set speed (17.6 mm/s)
  Call Extruder(211.58047)
  MoveL 5929 to (437.35, 515.73, 104) mm, rotated rx 180 ry 0 rz 160 deg; joints [9.499, 53.785, 15.084, -148.762, 71.713, 169.224]
  Set speed (17.6 mm/s)
  Call Extruder(215.35179)
  MoveL 5930 to (437.08, 514.59, 104) mm, rotated rx -180 ry 0 rz 160 deg; joints [9.34, 53.73, 15.206, -148.938, 71.742, 169.313]
  Set speed (17.6 mm/s)
  Call Extruder(220.78801)
  MoveL 5931 to (436.71, 512.94, 104) mm, rotated rx -180 ry 0 rz 160 deg; joints [9.11, 53.656, 15.374, -149.192, 71.779, 169.438]
  Set speed (17.6 mm/s)
  Call Extruder(228.69822)
  MoveL 5932 to (436.26, 510.51, 104) mm, rotated rx -180 ry 0 rz 160 deg; joints [8.768, 53.558, 15.593, -149.566, 71.822, 169.614]
  Set speed (17.6 mm/s)
  Call Extruder(237.15881)
  MoveL 5933 to (435.88, 507.89, 104) mm, rotated rx -180 ry 0 rz 160 deg; joints [8.396, 53.468, 15.797, -149.97, 71.854, 169.794]
  Set speed (17.6 mm/s)
  Call Extruder(245.61933)
  MoveL 5934 to (435.62, 505.26, 104) mm, rotated rx 180 ry 0 rz 160 deg; joints [8.018, 53.392, 15.968, -150.377, 71.87, 169.966]
  Set speed (17.6 mm/s)
  Call Extruder(253.90982)
  MoveL 5935 to (435.46, 502.68, 104) mm, rotated rx 180 ry 0 rz 160 deg; joints [7.644, 53.332, 16.104, -150.777, 71.871, 170.126]
  Call Extruder(262.45794)
  MoveL 5936 to (435.41, 500.01, 104) mm, rotated rx -180 ry 0 rz 160 deg; joints [7.254, 53.286, 16.209, -151.19, 71.856, 170.282]
  Set speed (17.6 mm/s)
  Call Extruder(270.15240)
  MoveL 5937 to (435.45, 497.61, 104) mm, rotated rx -180 ry 0 rz 160 deg; joints [6.901, 53.256, 16.277, -151.563, 71.83, 170.415]
  Call Extruder(277.60712)
  MoveL 5938 to (435.57, 495.28, 104) mm, rotated rx -180 ry 0 rz 160 deg; joints [6.557, 53.239, 16.316, -151.923, 71.793, 170.537]
  Call Extruder(285.21380)
  MoveL 5939 to (435.79, 492.92, 104) mm, rotated rx -180 ry 0 rz 160 deg; joints [6.206, 53.233, 16.329, -152.289, 71.742, 170.655]
  Set speed (17.6 mm/s)
  Call Extruder(292.88935)
  MoveL 5940 to (436.1, 490.54, 104) mm, rotated rx -180 ry 0 rz 160 deg; joints [5.851, 53.24, 16.314, -152.656, 71.677, 170.767]
  Set speed (17.6 mm/s)
  Call Extruder(300.43874)
  MoveL 5941 to (436.49, 488.21, 104) mm, rotated rx -180 ry 0 rz 160 deg; joints [5.503, 53.258, 16.273, -153.015, 71.601, 170.869]
  Set speed (17.6 mm/s)
  Call Extruder(308.34572)
  MoveL 5942 to (436.98, 485.79, 104) mm, rotated rx 180 ry 0 rz 160 deg; joints [5.14, 53.29, 16.2, -153.387, 71.508, 170.97]
  Set speed (17.6 mm/s)
  Call Extruder(315.73036)
  MoveL 5943 to (437.53, 483.55, 104) mm, rotated rx -180 ry 0 rz 160 deg; joints [4.804, 53.331, 16.107, -153.73, 71.408, 171.057]
  Call Extruder(323.34215)
  MoveL 5944 to (438.18, 481.26, 104) mm, rotated rx 180 ry 0 rz 160 deg; joints [4.46, 53.385, 15.984, -154.078, 71.294, 171.14]
  Set speed (17.6 mm/s)
  Call Extruder(330.95792)
  MoveL 5945 to (438.91, 479, 104) mm, rotated rx -180 ry 0 rz 160 deg; joints [4.119, 53.452, 15.834, -154.421, 71.166, 171.216]
  Call Extruder(338.59756)
  MoveL 5946 to (439.73, 476.76, 104) mm, rotated rx 180 ry 0 rz 160 deg; joints [3.782, 53.53, 15.658, -154.759, 71.026, 171.286]
  Set speed (17.6 mm/s)
  Call Extruder(346.26009)
  MoveL 5947 to (440.63, 474.54, 104) mm, rotated rx 180 ry 0 rz 160 deg; joints [3.448, 53.62, 15.455, -155.091, 70.873, 171.349]
  Set speed (17.6 mm/s)
  Call Extruder(353.78583)
  MoveL 5948 to (441.6, 472.39, 104) mm, rotated rx 180 ry 0 rz 160 deg; joints [3.127, 53.72, 15.229, -155.41, 70.711, 171.404]
  Call Extruder(361.48155)
  MoveL 5949 to (442.67, 470.24, 104) mm, rotated rx 180 ry 0 rz 160 deg; joints [2.804, 53.834, 14.973, -155.727, 70.533, 171.454]
  Set speed (17.6 mm/s)
  Call Extruder(369.01412)
  MoveL 5950 to (443.79, 468.17, 104) mm, rotated rx 180 ry 0 rz 160 deg; joints [2.495, 53.957, 14.697, -156.029, 70.348, 171.496]
  Set speed (17.6 mm/s)
  Call Extruder(376.66161)
  MoveL 5951 to (445, 466.11, 104) mm, rotated rx -180 ry 0 rz 160 deg; joints [2.189, 54.092, 14.392, -156.326, 70.148, 171.532]
  Set speed (17.6 mm/s)
  Call Extruder(384.24660)
  MoveL 5952 to (446.28, 464.12, 104) mm, rotated rx -180 ry 0 rz 160 deg; joints [1.893, 54.238, 14.065, -156.611, 69.938, 171.561]
  Set speed (17.6 mm/s)
  Call Extruder(391.75143)
  MoveL 5953 to (447.62, 462.19, 104) mm, rotated rx 180 ry 0 rz 160 deg; joints [1.609, 54.393, 13.719, -156.883, 69.721, 171.584]
  Set speed (17.6 mm/s)
  Call Extruder(399.45136)
  MoveL 5954 to (449.07, 460.27, 104) mm, rotated rx 180 ry 0 rz 160 deg; joints [1.327, 54.563, 13.338, -157.15, 69.486, 171.6]
  Set speed (17.6 mm/s)
  Call Extruder(406.99606)
  MoveL 5955 to (450.55, 458.44, 104) mm, rotated rx 180 ry 0 rz 160 deg; joints [1.059, 54.74, 12.943, -157.401, 69.246, 171.61]
  Call Extruder(414.76125)
  MoveL 5956 to (452.15, 456.61, 104) mm, rotated rx 180 ry 0 rz 160 deg; joints [0.794, 54.933, 12.514, -157.648, 68.988, 171.613]
  Call Extruder(422.37230)
  MoveL 5957 to (453.78, 454.88, 104) mm, rotated rx 180 ry 0 rz 160 deg; joints [0.545, 55.133, 12.071, -157.877, 68.726, 171.609]
  Set speed (17.6 mm/s)
  Call Extruder(429.80094)
  MoveL 5958 to (455.43, 453.25, 104) mm, rotated rx 180 ry 0 rz 160 deg; joints [0.312, 55.337, 11.617, -158.088, 68.462, 171.6]
  Set speed (17.6 mm/s)
  Call Extruder(437.50255)
  MoveL 5959 to (457.2, 451.62, 104) mm, rotated rx -180 ry 0 rz 160 deg; joints [0.081, 55.559, 11.127, -158.294, 68.178, 171.583]
  Call Extruder(445.20164)
  MoveL 5960 to (459.03, 450.06, 104) mm, rotated rx -180 ry 0 rz 160 deg; joints [-0.138, 55.79, 10.616, -158.486, 67.886, 171.559]
  Set speed (17.6 mm/s)
  Call Extruder(452.67033)
  MoveL 5961 to (460.86, 448.61, 104) mm, rotated rx 180 ry 0 rz 160 deg; joints [-0.34, 56.024, 10.1, -158.659, 67.594, 171.53]
  Set speed (17.6 mm/s)
  Call Extruder(460.43581)
  MoveL 5962 to (462.82, 447.18, 104) mm, rotated rx -180 ry 0 rz 160 deg; joints [-0.537, 56.276, 9.545, -158.825, 67.283, 171.492]
  Set speed (17.6 mm/s)
  Call Extruder(467.95109)
  MoveL 5963 to (464.76, 445.86, 104) mm, rotated rx 180 ry 0 rz 160 deg; joints [-0.717, 56.529, 8.991, -158.973, 66.975, 171.449]
  Set speed (17.6 mm/s)
  Call Extruder(475.64667)
  MoveL 5964 to (466.8, 444.59, 104) mm, rotated rx 180 ry 0 rz 160 deg; joints [-0.889, 56.796, 8.405, -159.108, 66.652, 171.398]
  Set speed (17.6 mm/s)
  Call Extruder(483.26375)
  MoveL 5965 to (468.86, 443.4, 104) mm, rotated rx 180 ry 0 rz 160 deg; joints [-1.047, 57.069, 7.808, -159.229, 66.325, 171.34]
  Set speed (17.6 mm/s)
  Call Extruder(491.82595)
  MoveL 5966 to (471.23, 442.16, 104) mm, rotated rx 180 ry 0 rz 160 deg; joints [-1.21, 57.386, 7.119, -159.346, 65.952, 171.267]
  Set speed (17.6 mm/s)
  Call Extruder(498.46697)
  MoveL 5967 to (473.1, 441.27, 104) mm, rotated rx 180 ry 0 rz 160 deg; joints [-1.326, 57.638, 6.57, -159.425, 65.657, 171.204]
  Set speed (17.6 mm/s)
  Call Extruder(506.12792)
  MoveL 5968 to (475.29, 440.31, 104) mm, rotated rx 180 ry 0 rz 160 deg; joints [-1.447, 57.936, 5.923, -159.501, 65.311, 171.125]
  Set speed (17.6 mm/s)
  Call Extruder(513.64387)
  MoveL 5969 to (477.48, 439.45, 104) mm, rotated rx 180 ry 0 rz 160 deg; joints [-1.556, 58.235, 5.274, -159.562, 64.967, 171.039]
  Set speed (17.6 mm/s)
  Call Extruder(521.30416)
  MoveL 5970 to (479.74, 438.66, 104) mm, rotated rx 180 ry 0 rz 160 deg; joints [-1.653, 58.548, 4.6, -159.609, 64.612, 170.945]
  Call Extruder(528.81532)
  MoveL 5971 to (481.98, 437.97, 104) mm, rotated rx 180 ry 0 rz 160 deg; joints [-1.737, 58.86, 3.926, -159.641, 64.261, 170.845]
  Set speed (17.6 mm/s)
  Call Extruder(536.47450)
  MoveL 5972 to (484.29, 437.34, 104) mm, rotated rx -180 ry 0 rz 160 deg; joints [-1.81, 59.185, 3.227, -159.658, 63.898, 170.736]
  Set speed (17.6 mm/s)
  Call Extruder(544.19809)
  MoveL 5973 to (486.64, 436.8, 104) mm, rotated rx 180 ry 0 rz 160 deg; joints [-1.871, 59.519, 2.511, -159.66, 63.53, 170.617]
  Set speed (17.6 mm/s)
  Call Extruder(551.72164)
  MoveL 5974 to (488.95, 436.35, 104) mm, rotated rx 180 ry 0 rz 160 deg; joints [-1.92, 59.849, 1.803, -159.648, 63.168, 170.495]
  Set speed (17.6 mm/s)
  Call Extruder(559.00005)
  MoveL 5975 to (491.19, 436, 104) mm, rotated rx 180 ry 0 rz 160 deg; joints [-1.955, 60.174, 1.11, -159.622, 62.816, 170.368]
  Set speed (17.6 mm/s)
  Call Extruder(566.99116)
  MoveL 5976 to (493.67, 435.71, 104) mm, rotated rx 180 ry 0 rz 160 deg; joints [-1.982, 60.535, 0.34, -159.577, 62.429, 170.222]
  Set speed (17.6 mm/s)
  Call Extruder(574.56145)
  MoveL 5977 to (496.03, 435.53, 104) mm, rotated rx 180 ry 0 rz 160 deg; joints [-1.996, 60.882, -0.398, -159.521, 62.06, 170.074]
  Set speed (17.6 mm/s)
  Call Extruder(582.25413)
  MoveL 5978 to (498.43, 435.42, 104) mm, rotated rx -180 ry 0 rz 160 deg; joints [-1.998, 61.239, -1.155, -159.449, 61.685, 169.917]
  Set speed (17.6 mm/s)
  Call Extruder(589.78974)
  MoveL 5979 to (500.79, 435.41, 104) mm, rotated rx 180 ry 0 rz 160 deg; joints [-1.99, 61.592, -1.903, -159.363, 61.316, 169.754]
  Set speed (17.6 mm/s)
  Call Extruder(597.27567)
  MoveL 5980 to (503.12, 435.48, 104) mm, rotated rx 180 ry 0 rz 160 deg; joints [-1.97, 61.946, -2.652, -159.265, 60.951, 169.584]
  Set speed (17.6 mm/s)
  Call Extruder(605.01041)
  MoveL 5981 to (505.54, 435.64, 104) mm, rotated rx -180 ry 0 rz 160 deg; joints [-1.94, 62.315, -3.43, -159.149, 60.574, 169.401]
  Set speed (17.6 mm/s)
  Call Extruder(612.46041)
  MoveL 5982 to (507.85, 435.88, 104) mm, rotated rx 180 ry 0 rz 160 deg; joints [-1.9, 62.672, -4.182, -159.024, 60.213, 169.216]
  Set speed (17.6 mm/s)
  Call Extruder(620.14270)
  MoveL 5983 to (510.23, 436.22, 104) mm, rotated rx 180 ry 0 rz 160 deg; joints [-1.848, 63.043, -4.961, -158.881, 59.841, 169.018]
  Set speed (17.6 mm/s)
  Call Extruder(627.85376)
  MoveL 5984 to (512.6, 436.64, 104) mm, rotated rx -180 ry 0 rz 160 deg; joints [-1.786, 63.417, -5.745, -158.723, 59.471, 168.811]
  Call Extruder(635.47545)
  MoveL 5985 to (514.93, 437.15, 104) mm, rotated rx 180 ry 0 rz 160 deg; joints [-1.714, 63.788, -6.521, -158.554, 59.108, 168.597]
  Call Extruder(642.95425)
  MoveL 5986 to (517.19, 437.73, 104) mm, rotated rx -180 ry 0 rz 160 deg; joints [-1.634, 64.152, -7.282, -158.375, 58.755, 168.38]
  Call Extruder(650.49262)
  MoveL 5987 to (519.45, 438.4, 104) mm, rotated rx 180 ry 0 rz 160 deg; joints [-1.545, 64.52, -8.049, -158.182, 58.403, 168.154]
  Set speed (17.6 mm/s)
  Call Extruder(658.15517)
  MoveL 5988 to (521.72, 439.17, 104) mm, rotated rx 180 ry 0 rz 160 deg; joints [-1.445, 64.894, -8.826, -157.973, 58.049, 167.916]
  Set speed (17.6 mm/s)
  Call Extruder(665.75476)
  MoveL 5989 to (523.94, 440, 104) mm, rotated rx -180 ry 0 rz 160 deg; joints [-1.336, 65.264, -9.595, -157.754, 57.703, 167.672]
  Set speed (17.6 mm/s)
  Call Extruder(673.34962)
  MoveL 5990 to (526.13, 440.92, 104) mm, rotated rx 180 ry 0 rz 160 deg; joints [-1.219, 65.632, -10.359, -157.523, 57.362, 167.421]
  Set speed (17.6 mm/s)
  Call Extruder(681.18597)
  MoveL 5991 to (528.35, 441.96, 104) mm, rotated rx 180 ry 0 rz 160 deg; joints [-1.09, 66.011, -11.143, -157.272, 57.016, 167.154]
  Call Extruder(688.63720)
  MoveL 5992 to (530.42, 443.01, 104) mm, rotated rx 180 ry 0 rz 160 deg; joints [-0.959, 66.37, -11.883, -157.023, 56.694, 166.894]
  Set speed (17.6 mm/s)
  Call Extruder(696.39830)
  MoveL 5993 to (532.54, 444.2, 104) mm, rotated rx 180 ry 0 rz 160 deg; joints [-0.814, 66.74, -12.647, -156.752, 56.365, 166.615]
  Set speed (17.6 mm/s)
  Call Extruder(703.80802)
  MoveL 5994 to (534.52, 445.4, 104) mm, rotated rx -180 ry 0 rz 160 deg; joints [-0.668, 67.091, -13.37, -156.483, 56.058, 166.343]
  Call Extruder(711.62019)
  MoveL 5995 to (536.56, 446.74, 104) mm, rotated rx -180 ry 0 rz 160 deg; joints [-0.507, 67.457, -14.123, -156.189, 55.742, 166.049]
  Set speed (17.6 mm/s)
  Call Extruder(719.14817)
  MoveL 5996 to (538.47, 448.11, 104) mm, rotated rx 180 ry 0 rz 160 deg; joints [-0.345, 67.806, -14.838, -155.895, 55.446, 165.761]
  Call Extruder(726.64901)
  MoveL 5997 to (540.33, 449.54, 104) mm, rotated rx -180 ry 0 rz 160 deg; joints [-0.176, 68.149, -15.541, -155.594, 55.16, 165.468]
  Set speed (17.6 mm/s)
  Call Extruder(734.30436)
  MoveL 5998 to (542.17, 451.07, 104) mm, rotated rx -180 ry 0 rz 160 deg; joints [0.003, 68.493, -16.246, -155.278, 54.878, 165.164]
  Set speed (17.6 mm/s)
  Call Extruder(742.06489)
  MoveL 5999 to (543.98, 452.68, 104) mm, rotated rx 180 ry 0 rz 160 deg; joints [0.19, 68.836, -16.948, -154.95, 54.601, 164.851]
  Set speed (17.6 mm/s)
  Call Extruder(749.54369)
  MoveL 6000 to (545.66, 454.31, 104) mm, rotated rx -180 ry 0 rz 160 deg; joints [0.378, 69.161, -17.61, -154.625, 54.344, 164.545]
  Call Extruder(753.73854)
  MoveL 6001 to (546.58, 455.24, 104) mm, rotated rx 180 ry 0 rz 160 deg; joints [0.485, 69.34, -17.976, -154.44, 54.205, 164.372]
  Call Extruder(757.97600)
  MoveL 6002 to (547.48, 456.21, 104) mm, rotated rx 180 ry 0 rz 160 deg; joints [0.595, 69.519, -18.34, -154.251, 54.068, 164.196]
  Set speed (17.6 mm/s)
  Call Extruder(762.59413)
  MoveL 6003 to (548.45, 457.28, 104) mm, rotated rx 180 ry 0 rz 160 deg; joints [0.718, 69.711, -18.731, -154.042, 53.922, 164.004]
  Set speed (17.6 mm/s)
  Call Extruder(766.46745)
  MoveL 6004 to (549.24, 458.19, 104) mm, rotated rx 180 ry 0 rz 160 deg; joints [0.821, 69.87, -19.054, -153.866, 53.803, 163.841]
  Set speed (17.6 mm/s)
  Call Extruder(770.68757)
  MoveL 6005 to (550.08, 459.21, 104) mm, rotated rx -180 ry 0 rz 160 deg; joints [0.937, 70.04, -19.4, -153.672, 53.678, 163.664]
  Set speed (17.6 mm/s)
  Call Extruder(775.27196)
  MoveL 6006 to (550.98, 460.32, 104) mm, rotated rx 180 ry 0 rz 160 deg; joints [1.063, 70.222, -19.771, -153.46, 53.545, 163.47]
  Set speed (17.6 mm/s)
  Call Extruder(779.49139)
  MoveL 6007 to (551.78, 461.37, 104) mm, rotated rx -180 ry 0 rz 160 deg; joints [1.181, 70.387, -20.106, -153.262, 53.426, 163.291]
  Call Extruder(783.38711)
  MoveL 6008 to (552.5, 462.36, 104) mm, rotated rx 180 ry 0 rz 160 deg; joints [1.292, 70.537, -20.41, -153.079, 53.321, 163.126]
  Set speed (17.6 mm/s)
  Call Extruder(788.01362)
  MoveL 6009 to (553.32, 463.54, 104) mm, rotated rx 180 ry 0 rz 160 deg; joints [1.424, 70.711, -20.764, -152.86, 53.2, 162.93]
  Set speed (17.6 mm/s)
  Call Extruder(791.89502)
  MoveL 6010 to (554, 464.55, 104) mm, rotated rx -180 ry 0 rz 160 deg; joints [1.537, 70.855, -21.055, -152.674, 53.102, 162.765]
  Call Extruder(796.50700)
  MoveL 6011 to (554.78, 465.76, 104) mm, rotated rx -180 ry 0 rz 160 deg; joints [1.672, 71.022, -21.393, -152.453, 52.99, 162.569]
  Set speed (17.6 mm/s)
  Call Extruder(800.25528)
  MoveL 6012 to (555.39, 466.76, 104) mm, rotated rx 180 ry 0 rz 160 deg; joints [1.784, 71.155, -21.663, -152.273, 52.903, 162.409]
  Call Extruder(804.54695)
  MoveL 6013 to (556.07, 467.92, 104) mm, rotated rx 180 ry 0 rz 160 deg; joints [1.912, 71.304, -21.964, -152.065, 52.807, 162.227]
  Set speed (17.6 mm/s)
  Call Extruder(810.03074)
  MoveL 6014 to (556.9, 469.41, 104) mm, rotated rx 180 ry 0 rz 160 deg; joints [2.078, 71.489, -22.339, -151.799, 52.691, 161.995]
  Call Extruder(813.07217)
  MoveL 6015 to (557.34, 470.25, 104) mm, rotated rx 180 ry 0 rz 160 deg; joints [2.172, 71.588, -22.54, -151.65, 52.63, 161.867]
  Set speed (17.6 mm/s)
  Call Extruder(817.24649)
  MoveL 6016 to (557.93, 471.42, 104) mm, rotated rx 180 ry 0 rz 160 deg; joints [2.3, 71.723, -22.811, -151.447, 52.55, 161.691]
  Set speed (17.6 mm/s)
  Call Extruder(822.70708)
  MoveL 6017 to (558.66, 472.95, 104) mm, rotated rx 180 ry 0 rz 160 deg; joints [2.47, 71.893, -23.154, -151.18, 52.452, 161.463]
  Set speed (17.6 mm/s)
  Call Extruder(825.64659)
  MoveL 6018 to (559.04, 473.79, 104) mm, rotated rx 180 ry 0 rz 160 deg; joints [2.562, 71.981, -23.333, -151.036, 52.402, 161.34]
  Set speed (17.6 mm/s)
  Call Extruder(834.05572)
  MoveL 6019 to (560.06, 476.21, 104) mm, rotated rx 180 ry 0 rz 160 deg; joints [2.829, 72.224, -23.823, -150.624, 52.272, 160.993]
  Set speed (17.6 mm/s)
  Call Extruder(838.43005)
  MoveL 6020 to (560.54, 477.49, 104) mm, rotated rx 180 ry 0 rz 160 deg; joints [2.969, 72.343, -24.063, -150.41, 52.213, 160.815]
  Call Extruder(842.52163)
  MoveL 6021 to (560.98, 478.69, 104) mm, rotated rx -180 ry 0 rz 160 deg; joints [3.101, 72.452, -24.283, -150.21, 52.16, 160.649]
  Call Extruder(846.90956)
  MoveL 6022 to (561.41, 479.99, 104) mm, rotated rx -180 ry 0 rz 160 deg; joints [3.244, 72.562, -24.505, -149.996, 52.111, 160.474]
  Set speed (17.6 mm/s)
  Call Extruder(851.07662)
  MoveL 6023 to (561.81, 481.22, 104) mm, rotated rx 180 ry 0 rz 160 deg; joints [3.379, 72.665, -24.711, -149.794, 52.066, 160.309]
  Set speed (17.6 mm/s)
  Call Extruder(855.37325)
  MoveL 6024 to (562.18, 482.51, 104) mm, rotated rx 180 ry 0 rz 160 deg; joints [3.521, 72.764, -24.911, -149.586, 52.028, 160.141]
  Set speed (17.6 mm/s)
  Call Extruder(859.52345)
  MoveL 6025 to (562.52, 483.76, 104) mm, rotated rx 180 ry 0 rz 160 deg; joints [3.657, 72.857, -25.098, -149.385, 51.993, 159.98]
  Set speed (17.6 mm/s)
  Call Extruder(863.85607)
  MoveL 6026 to (562.84, 485.07, 104) mm, rotated rx -180 ry 0 rz 160 deg; joints [3.801, 72.947, -25.279, -149.177, 51.964, 159.815]
  Set speed (17.6 mm/s)
  Call Extruder(867.97610)
  MoveL 6027 to (563.13, 486.32, 104) mm, rotated rx 180 ry 0 rz 160 deg; joints [3.939, 73.03, -25.447, -148.98, 51.939, 159.659]
  Set speed (17.6 mm/s)
  Call Extruder(876.52953)
  MoveL 6028 to (563.65, 488.95, 104) mm, rotated rx 180 ry 0 rz 160 deg; joints [4.226, 73.187, -25.762, -148.573, 51.905, 159.344]
  Set speed (17.6 mm/s)
  Call Extruder(884.97152)
  MoveL 6029 to (564.04, 491.55, 104) mm, rotated rx 180 ry 0 rz 160 deg; joints [4.512, 73.321, -26.032, -148.178, 51.891, 159.044]
  Call Extruder(893.53431)
  MoveL 6030 to (564.34, 494.21, 104) mm, rotated rx -180 ry 0 rz 160 deg; joints [4.804, 73.436, -26.263, -147.783, 51.897, 158.752]
  Set speed (17.6 mm/s)
  Call Extruder(901.89298)
  MoveL 6031 to (564.52, 496.82, 104) mm, rotated rx -180 ry 0 rz 160 deg; joints [5.091, 73.529, -26.449, -147.405, 51.923, 158.479]
  Set speed (17.6 mm/s)
  Call Extruder(910.34197)
  MoveL 6032 to (564.6, 499.46, 104) mm, rotated rx -180 ry 0 rz 160 deg; joints [5.382, 73.601, -26.594, -147.03, 51.97, 158.217]
  Set speed (17.6 mm/s)
  Call Extruder(918.66811)
  MoveL 6033 to (564.56, 502.06, 104) mm, rotated rx -180 ry 0 rz 160 deg; joints [5.67, 73.651, -26.695, -146.67, 52.034, 157.973]
  Set speed (17.6 mm/s)
  Call Extruder(927.24047)
  MoveL 6034 to (564.43, 504.74, 104) mm, rotated rx 180 ry 0 rz 160 deg; joints [5.967, 73.682, -26.756, -146.308, 52.121, 157.738]
  Set speed (17.6 mm/s)
  Call Extruder(935.61908)
  MoveL 6035 to (564.18, 507.34, 104) mm, rotated rx 180 ry 0 rz 160 deg; joints [6.257, 73.689, -26.771, -145.965, 52.225, 157.524]
  Set speed (17.6 mm/s)
  Call Extruder(944.25835)
  MoveL 6036 to (563.82, 510.02, 104) mm, rotated rx 180 ry 0 rz 160 deg; joints [6.557, 73.675, -26.742, -145.621, 52.352, 157.32]
  Set speed (17.6 mm/s)
  Call Extruder(952.51960)
  MoveL 6037 to (563.36, 512.56, 104) mm, rotated rx -180 ry 0 rz 160 deg; joints [6.843, 73.64, -26.672, -145.304, 52.491, 157.143]
  Set speed (17.6 mm/s)
  Call Extruder(961.13032)
  MoveL 6038 to (562.79, 515.19, 104) mm, rotated rx 180 ry 0 rz 160 deg; joints [7.14, 73.582, -26.556, -144.985, 52.655, 156.975]
  Set speed (17.6 mm/s)
  Call Extruder(965.33613)
  MoveL 6039 to (562.46, 516.46, 104) mm, rotated rx -180 ry 0 rz 160 deg; joints [7.284, 73.545, -26.481, -144.834, 52.743, 156.901]
  Call Extruder(969.55810)
  MoveL 6040 to (562.12, 517.73, 104) mm, rotated rx 180 ry 0 rz 160 deg; joints [7.429, 73.504, -26.399, -144.685, 52.833, 156.829]
  Set speed (17.6 mm/s)
  Call Extruder(977.89894)
  MoveL 6041 to (561.35, 520.22, 104) mm, rotated rx 180 ry 0 rz 160 deg; joints [7.715, 73.406, -26.203, -144.399, 53.026, 156.702]
  Set speed (17.6 mm/s)
  Call Extruder(982.24395)
  MoveL 6042 to (560.91, 521.5, 104) mm, rotated rx 180 ry 0 rz 160 deg; joints [7.863, 73.346, -26.082, -144.256, 53.134, 156.645]
  Call Extruder(986.38815)
  MoveL 6043 to (560.47, 522.72, 104) mm, rotated rx 180 ry 0 rz 160 deg; joints [8.004, 73.286, -25.961, -144.121, 53.239, 156.593]
  Set speed (17.6 mm/s)
  Call Extruder(990.71862)
  MoveL 6044 to (559.98, 523.98, 104) mm, rotated rx 180 ry 0 rz 160 deg; joints [8.15, 73.216, -25.82, -143.984, 53.355, 156.544]
  Set speed (17.6 mm/s)
  Call Extruder(994.90643)
  MoveL 6045 to (559.49, 525.19, 104) mm, rotated rx 180 ry 0 rz 160 deg; joints [8.292, 73.145, -25.678, -143.854, 53.469, 156.5]
  Call Extruder(999.18662)
  MoveL 6046 to (558.94, 526.41, 104) mm, rotated rx 180 ry 0 rz 160 deg; joints [8.436, 73.065, -25.518, -143.725, 53.591, 156.462]
  Set speed (17.6 mm/s)
  Call Extruder(1003.22306)
  MoveL 6047 to (558.42, 527.56, 104) mm, rotated rx -180 ry 0 rz 160 deg; joints [8.571, 72.988, -25.363, -143.605, 53.708, 156.428]
  Call Extruder(1006.42473)
  MoveL 6048 to (557.99, 528.46, 104) mm, rotated rx -180 ry 0 rz 160 deg; joints [8.677, 72.923, -25.232, -143.513, 53.804, 156.405]
  Call Extruder(1011.78326)
  MoveL 6049 to (557.23, 529.95, 104) mm, rotated rx 180 ry 0 rz 160 deg; joints [8.855, 72.807, -24.998, -143.362, 53.969, 156.373]
  Set speed (17.6 mm/s)
  Call Extruder(1016.09643)
  MoveL 6050 to (556.6, 531.14, 104) mm, rotated rx 180 ry 0 rz 160 deg; joints [8.997, 72.709, -24.8, -143.244, 54.106, 156.352]
  Set speed (17.6 mm/s)
  Call Extruder(1020.26087)
  MoveL 6051 to (555.96, 532.27, 104) mm, rotated rx 180 ry 0 rz 160 deg; joints [9.134, 72.609, -24.599, -143.134, 54.242, 156.336]
  Call Extruder(1024.45972)
  MoveL 6052 to (555.29, 533.41, 104) mm, rotated rx 180 ry 0 rz 160 deg; joints [9.271, 72.505, -24.389, -143.025, 54.381, 156.324]
  Set speed (17.6 mm/s)
  Call Extruder(1029.13445)
  MoveL 6053 to (554.52, 534.65, 104) mm, rotated rx -180 ry 0 rz 160 deg; joints [9.422, 72.383, -24.143, -142.908, 54.541, 156.317]
  Set speed (17.6 mm/s)
  Call Extruder(1032.94523)
  MoveL 6054 to (553.87, 535.64, 104) mm, rotated rx -180 ry 0 rz 160 deg; joints [9.545, 72.28, -23.936, -142.815, 54.674, 156.315]
  Set speed (17.6 mm/s)
  Call Extruder(1037.12875)
  MoveL 6055 to (553.14, 536.73, 104) mm, rotated rx 180 ry 0 rz 160 deg; joints [9.678, 72.162, -23.699, -142.716, 54.822, 156.317]
  Call Extruder(1041.44229)
  MoveL 6056 to (552.36, 537.83, 104) mm, rotated rx 180 ry 0 rz 160 deg; joints [9.815, 72.038, -23.447, -142.617, 54.978, 156.323]
  Set speed (17.6 mm/s)
  Call Extruder(1045.60295)
  MoveL 6057 to (551.59, 538.88, 104) mm, rotated rx 180 ry 0 rz 160 deg; joints [9.946, 71.913, -23.196, -142.525, 55.132, 156.333]
  Set speed (17.6 mm/s)
  Call Extruder(1049.92109)
  MoveL 6058 to (550.77, 539.95, 104) mm, rotated rx 180 ry 0 rz 160 deg; joints [10.081, 71.78, -22.927, -142.432, 55.293, 156.348]
  Set speed (17.6 mm/s)
  Call Extruder(1054.06933)
  MoveL 6059 to (549.96, 540.96, 104) mm, rotated rx -180 ry 0 rz 160 deg; joints [10.21, 71.648, -22.661, -142.345, 55.451, 156.366]
  Set speed (17.6 mm/s)
  Call Extruder(1058.29433)
  MoveL 6060 to (549.11, 541.97, 104) mm, rotated rx -180 ry 0 rz 160 deg; joints [10.339, 71.51, -22.381, -142.261, 55.615, 156.389]
  Set speed (17.6 mm/s)
  Call Extruder(1062.17816)
  MoveL 6061 to (548.31, 542.88, 104) mm, rotated rx 180 ry 0 rz 160 deg; joints [10.457, 71.38, -22.118, -142.185, 55.768, 156.414]
  Set speed (17.6 mm/s)
  Call Extruder(1066.74397)
  MoveL 6062 to (547.35, 543.94, 104) mm, rotated rx -180 ry 0 rz 160 deg; joints [10.595, 71.224, -21.803, -142.099, 55.949, 156.447]
  Set speed (17.6 mm/s)
  Call Extruder(1070.54808)
  MoveL 6063 to (546.53, 544.81, 104) mm, rotated rx -180 ry 0 rz 160 deg; joints [10.709, 71.09, -21.532, -142.03, 56.102, 156.478]
  Set speed (17.6 mm/s)
  Call Extruder(1075.22295)
  MoveL 6064 to (545.51, 545.85, 104) mm, rotated rx 180 ry 0 rz 160 deg; joints [10.847, 70.922, -21.192, -141.949, 56.293, 156.521]
  Set speed (17.6 mm/s)
  Call Extruder(1078.67396)
  MoveL 6065 to (544.74, 546.6, 104) mm, rotated rx 180 ry 0 rz 160 deg; joints [10.947, 70.796, -20.936, -141.891, 56.435, 156.556]
  Set speed (17.6 mm/s)
  Call Extruder(1084.55212)
  MoveL 6066 to (543.4, 547.85, 104) mm, rotated rx 180 ry 0 rz 160 deg; joints [11.117, 70.576, -20.491, -141.797, 56.68, 156.621]
  Set speed (17.6 mm/s)
  Call Extruder(1088.31360)
  MoveL 6067 to (542.52, 548.63, 104) mm, rotated rx -180 ry 0 rz 160 deg; joints [11.223, 70.433, -20.198, -141.74, 56.839, 156.666]
  Set speed (17.6 mm/s)
  Call Extruder(1092.13992)
  MoveL 6068 to (541.61, 549.41, 104) mm, rotated rx -180 ry 0 rz 160 deg; joints [11.331, 70.284, -19.897, -141.684, 57.001, 156.715]
  Set speed (17.6 mm/s)
  Call Extruder(1096.41253)
  MoveL 6069 to (540.58, 550.26, 104) mm, rotated rx 180 ry 0 rz 160 deg; joints [11.45, 70.115, -19.554, -141.624, 57.185, 156.773]
  Call Extruder(1100.65577)
  MoveL 6070 to (539.54, 551.08, 104) mm, rotated rx -180 ry 0 rz 160 deg; joints [11.566, 69.945, -19.207, -141.567, 57.368, 156.834]
  Set speed (17.6 mm/s)
  Call Extruder(1104.93713)
  MoveL 6071 to (538.48, 551.89, 104) mm, rotated rx -180 ry 0 rz 160 deg; joints [11.681, 69.77, -18.852, -141.513, 57.555, 156.9]
  Set speed (17.6 mm/s)
  Call Extruder(1109.04009)
  MoveL 6072 to (537.44, 552.64, 104) mm, rotated rx 180 ry 0 rz 160 deg; joints [11.791, 69.601, -18.507, -141.463, 57.735, 156.966]
  Call Extruder(1113.28540)
  MoveL 6073 to (536.35, 553.4, 104) mm, rotated rx 180 ry 0 rz 160 deg; joints [11.902, 69.423, -18.145, -141.415, 57.923, 157.037]
  Call Extruder(1117.47298)
  MoveL 6074 to (535.26, 554.12, 104) mm, rotated rx -180 ry 0 rz 160 deg; joints [12.01, 69.245, -17.783, -141.369, 58.109, 157.11]
  Set speed (17.6 mm/s)
  Call Extruder(1121.85884)
  MoveL 6075 to (534.11, 554.86, 104) mm, rotated rx -180 ry 0 rz 160 deg; joints [12.121, 69.057, -17.398, -141.325, 58.306, 157.191]
  Call Extruder(1126.01998)
  MoveL 6076 to (532.99, 555.53, 104) mm, rotated rx -180 ry 0 rz 160 deg; joints [12.225, 68.876, -17.028, -141.285, 58.493, 157.271]
  Set speed (17.6 mm/s)
  Call Extruder(1130.30082)
  MoveL 6077 to (531.84, 556.21, 104) mm, rotated rx 180 ry 0 rz 160 deg; joints [12.33, 68.688, -16.645, -141.246, 58.686, 157.355]
  Set speed (17.6 mm/s)
  Call Extruder(1133.85426)
  MoveL 6078 to (530.87, 556.75, 104) mm, rotated rx 180 ry 0 rz 160 deg; joints [12.415, 68.53, -16.322, -141.216, 58.848, 157.428]
  Set speed (17.6 mm/s)
  Call Extruder(1139.90934)
  MoveL 6079 to (529.2, 557.63, 104) mm, rotated rx 180 ry 0 rz 160 deg; joints [12.558, 68.259, -15.768, -141.17, 59.123, 157.556]
  Set speed (17.6 mm/s)
  Call Extruder(1142.92670)
  MoveL 6080 to (528.35, 558.04, 104) mm, rotated rx -180 ry 0 rz 160 deg; joints [12.627, 68.123, -15.488, -141.149, 59.261, 157.622]
  Set speed (17.6 mm/s)
  Call Extruder(1147.25392)
  MoveL 6081 to (527.13, 558.62, 104) mm, rotated rx 180 ry 0 rz 160 deg; joints [12.725, 67.925, -15.083, -141.121, 59.46, 157.72]
  Set speed (17.6 mm/s)
  Call Extruder(1151.43287)
  MoveL 6082 to (525.94, 559.16, 104) mm, rotated rx -180 ry 0 rz 160 deg; joints [12.817, 67.733, -14.688, -141.097, 59.652, 157.818]
  Set speed (17.6 mm/s)
  Call Extruder(1155.65261)
  MoveL 6083 to (524.73, 559.68, 104) mm, rotated rx -180 ry 0 rz 160 deg; joints [12.908, 67.538, -14.289, -141.074, 59.846, 157.917]
  Set speed (17.6 mm/s)
  Call Extruder(1159.90222)
  MoveL 6084 to (523.5, 560.16, 104) mm, rotated rx 180 ry 0 rz 160 deg; joints [12.997, 67.339, -13.881, -141.055, 60.042, 158.022]
  Call Extruder(1164.15163)
  MoveL 6085 to (522.26, 560.64, 104) mm, rotated rx -180 ry 0 rz 160 deg; joints [13.085, 67.141, -13.473, -141.037, 60.238, 158.127]
  Call Extruder(1168.42670)
  MoveL 6086 to (521, 561.08, 104) mm, rotated rx 180 ry 0 rz 160 deg; joints [13.169, 66.939, -13.057, -141.023, 60.436, 158.237]
  Set speed (17.6 mm/s)
  Call Extruder(1172.48502)
  MoveL 6087 to (519.8, 561.49, 104) mm, rotated rx 180 ry 0 rz 160 deg; joints [13.249, 66.747, -12.662, -141.01, 60.623, 158.342]
  Set speed (17.6 mm/s)
  Call Extruder(1177.75944)
  MoveL 6088 to (518.23, 561.97, 104) mm, rotated rx 180 ry 0 rz 160 deg; joints [13.348, 66.496, -12.145, -140.999, 60.866, 158.483]
  Set speed (17.6 mm/s)
  Call Extruder(1180.92459)
  MoveL 6089 to (517.28, 562.24, 104) mm, rotated rx -180 ry 0 rz 160 deg; joints [13.406, 66.345, -11.833, -140.993, 61.012, 158.568]
  Set speed (17.6 mm/s)
  Call Extruder(1184.76212)
  MoveL 6090 to (516.12, 562.55, 104) mm, rotated rx 180 ry 0 rz 160 deg; joints [13.473, 66.161, -11.452, -140.989, 61.19, 158.675]
  Set speed (17.6 mm/s)
  Call Extruder(1189.41347)
  MoveL 6091 to (514.72, 562.9, 104) mm, rotated rx -180 ry 0 rz 160 deg; joints [13.554, 65.937, -10.99, -140.986, 61.404, 158.805]
  Set speed (17.6 mm/s)
  Call Extruder(1198.01159)
  MoveL 6092 to (512.09, 563.46, 104) mm, rotated rx 180 ry 0 rz 160 deg; joints [13.693, 65.521, -10.129, -140.99, 61.8, 159.053]
  Call Extruder(1206.52981)
  MoveL 6093 to (509.47, 563.9, 104) mm, rotated rx 180 ry 0 rz 160 deg; joints [13.821, 65.108, -9.271, -141.003, 62.191, 159.306]
  Set speed (17.6 mm/s)
  Call Extruder(1214.90425)
  MoveL 6094 to (506.87, 564.23, 104) mm, rotated rx -180 ry 0 rz 160 deg; joints [13.936, 64.699, -8.422, -141.027, 62.574, 159.563]
  Set speed (17.6 mm/s)
  Call Extruder(1223.40557)
  MoveL 6095 to (504.22, 564.46, 104) mm, rotated rx 180 ry 0 rz 160 deg; joints [14.041, 64.285, -7.558, -141.061, 62.96, 159.83]
  Set speed (17.6 mm/s)
  Call Extruder(1231.90965)
  MoveL 6096 to (501.57, 564.58, 104) mm, rotated rx -180 ry 0 rz 160 deg; joints [14.135, 63.87, -6.693, -141.106, 63.342, 160.102]
  Set speed (17.6 mm/s)
  Call Extruder(1240.20330)
  MoveL 6097 to (498.98, 564.59, 104) mm, rotated rx -180 ry 0 rz 160 deg; joints [14.214, 63.467, -5.849, -141.16, 63.712, 160.374]
  Set speed (10.0 mm/s)
  MoveL 6098 to (498.98, 564.59, 108) mm, rotated rx -180 ry 0 rz 160 deg; joints [14.214, 62.84, -5.574, -141.05, 63.438, 160.127]
  Set speed (120.0 mm/s)
  MoveL 6099 to (498.98, 563.49, 108) mm, rotated rx -180 ry 0 rz 160 deg; joints [14.083, 62.796, -5.484, -141.203, 63.43, 160.222]
  Set speed (17.1 mm/s)
  Call Extruder(1248.86178)
  MoveL 6100 to (496.36, 563.4, 108) mm, rotated rx -180 ry 0 rz 160 deg; joints [14.15, 62.388, -4.633, -141.269, 63.798, 160.499]
  Set speed (17.1 mm/s)
  Call Extruder(1257.46587)
  MoveL 6101 to (493.76, 563.2, 108) mm, rotated rx -180 ry 0 rz 160 deg; joints [14.205, 61.984, -3.79, -141.346, 64.159, 160.779]
  Set speed (17.1 mm/s)
  Call Extruder(1265.98978)
  MoveL 6102 to (491.2, 562.89, 108) mm, rotated rx 180 ry 0 rz 160 deg; joints [14.247, 61.587, -2.959, -141.432, 64.511, 161.061]
  Set speed (17.1 mm/s)
  Call Extruder(1274.46110)
  MoveL 6103 to (488.67, 562.48, 108) mm, rotated rx -180 ry 0 rz 160 deg; joints [14.276, 61.195, -2.137, -141.528, 64.857, 161.344]
  Set speed (17.1 mm/s)
  Call Extruder(1283.25545)
  MoveL 6104 to (486.06, 561.95, 108) mm, rotated rx 180 ry 0 rz 160 deg; joints [14.293, 60.791, -1.289, -141.639, 65.211, 161.641]
  Set speed (17.1 mm/s)
  Call Extruder(1287.49678)
  MoveL 6105 to (484.82, 561.65, 108) mm, rotated rx 180 ry 0 rz 160 deg; joints [14.295, 60.598, -0.883, -141.698, 65.378, 161.786]
  Set speed (17.0 mm/s)
  Call Extruder(1291.63361)
  MoveL 6106 to (483.61, 561.35, 108) mm, rotated rx 180 ry 0 rz 160 deg; joints [14.295, 60.411, -0.489, -141.756, 65.541, 161.927]
  Set speed (17.0 mm/s)
  Call Extruder(1296.03747)
  MoveL 6107 to (482.33, 560.99, 108) mm, rotated rx 180 ry 0 rz 160 deg; joints [14.291, 60.213, -0.072, -141.822, 65.712, 162.078]
  Call Extruder(1300.27592)
  MoveL 6108 to (481.1, 560.62, 108) mm, rotated rx -180 ry 0 rz 160 deg; joints [14.285, 60.024, 0.328, -141.887, 65.875, 162.223]
  Set speed (17.0 mm/s)
  Call Extruder(1304.64916)
  MoveL 6109 to (479.84, 560.21, 108) mm, rotated rx 180 ry 0 rz 160 deg; joints [14.273, 59.83, 0.738, -141.959, 66.042, 162.373]
  Set speed (17.1 mm/s)
  Call Extruder(1308.88351)
  MoveL 6110 to (478.63, 559.8, 108) mm, rotated rx 180 ry 0 rz 160 deg; joints [14.26, 59.644, 1.132, -142.029, 66.202, 162.519]
  Call Extruder(1313.29333)
  MoveL 6111 to (477.38, 559.33, 108) mm, rotated rx -180 ry 0 rz 160 deg; joints [14.241, 59.451, 1.541, -142.107, 66.366, 162.672]
  Set speed (17.0 mm/s)
  Call Extruder(1317.76585)
  MoveL 6112 to (476.12, 558.84, 108) mm, rotated rx 180 ry 0 rz 160 deg; joints [14.22, 59.257, 1.952, -142.187, 66.532, 162.826]
  Set speed (17.1 mm/s)
  Call Extruder(1324.99410)
  MoveL 6113 to (474.12, 557.99, 108) mm, rotated rx 180 ry 0 rz 160 deg; joints [14.176, 58.947, 2.61, -142.325, 66.794, 163.077]
  Set speed (17.1 mm/s)
  Call Extruder(1330.39340)
  MoveL 6114 to (472.63, 557.3, 108) mm, rotated rx -180 ry 0 rz 160 deg; joints [14.136, 58.718, 3.097, -142.434, 66.987, 163.264]
  Set speed (17.1 mm/s)
  Call Extruder(1334.69101)
  MoveL 6115 to (471.47, 556.73, 108) mm, rotated rx -180 ry 0 rz 160 deg; joints [14.1, 58.538, 3.48, -142.523, 67.138, 163.413]
  Set speed (17.1 mm/s)
  Call Extruder(1339.64937)
  MoveL 6116 to (470.13, 556.04, 108) mm, rotated rx -180 ry 0 rz 160 deg; joints [14.055, 58.333, 3.919, -142.63, 67.31, 163.585]
  Call Extruder(1343.30610)
  MoveL 6117 to (469.16, 555.51, 108) mm, rotated rx 180 ry 0 rz 160 deg; joints [14.018, 58.182, 4.24, -142.711, 67.436, 163.712]
  Set speed (17.1 mm/s)
  Call Extruder(1347.56165)
  MoveL 6118 to (468.04, 554.88, 108) mm, rotated rx -180 ry 0 rz 160 deg; joints [13.972, 58.01, 4.61, -142.809, 67.579, 163.859]
  Set speed (17.1 mm/s)
  Call Extruder(1351.79216)
  MoveL 6119 to (466.94, 554.22, 108) mm, rotated rx -180 ry 0 rz 160 deg; joints [13.922, 57.839, 4.974, -142.908, 67.72, 164.005]
  Call Extruder(1356.15025)
  MoveL 6120 to (465.82, 553.52, 108) mm, rotated rx -180 ry 0 rz 160 deg; joints [13.867, 57.666, 5.345, -143.014, 67.863, 164.155]
  Set speed (17.1 mm/s)
  Call Extruder(1360.39641)
  MoveL 6121 to (464.75, 552.82, 108) mm, rotated rx -180 ry 0 rz 160 deg; joints [13.81, 57.5, 5.702, -143.12, 68, 164.302]
  Set speed (17.1 mm/s)
  Call Extruder(1364.69117)
  MoveL 6122 to (463.67, 552.08, 108) mm, rotated rx -180 ry 0 rz 160 deg; joints [13.749, 57.333, 6.059, -143.23, 68.136, 164.449]
  Set speed (17.1 mm/s)
  Call Extruder(1369.06164)
  MoveL 6123 to (462.6, 551.32, 108) mm, rotated rx 180 ry 0 rz 160 deg; joints [13.683, 57.166, 6.419, -143.344, 68.273, 164.598]
  Set speed (17.1 mm/s)
  Call Extruder(1373.83848)
  MoveL 6124 to (461.44, 550.45, 108) mm, rotated rx 180 ry 0 rz 160 deg; joints [13.606, 56.986, 6.807, -143.473, 68.419, 164.76]
  Set speed (17.1 mm/s)
  Call Extruder(1376.84911)
  MoveL 6125 to (460.72, 549.89, 108) mm, rotated rx -180 ry 0 rz 160 deg; joints [13.555, 56.874, 7.048, -143.556, 68.51, 164.863]
  Set speed (17.1 mm/s)
  Call Extruder(1381.25162)
  MoveL 6126 to (459.68, 549.06, 108) mm, rotated rx 180 ry 0 rz 160 deg; joints [13.478, 56.712, 7.397, -143.68, 68.641, 165.011]
  Set speed (17.1 mm/s)
  Call Extruder(1386.20287)
  MoveL 6127 to (458.53, 548.1, 108) mm, rotated rx 180 ry 0 rz 160 deg; joints [13.386, 56.533, 7.784, -143.823, 68.785, 165.177]
  Set speed (17.1 mm/s)
  Call Extruder(1390.50105)
  MoveL 6128 to (457.56, 547.23, 108) mm, rotated rx 180 ry 0 rz 160 deg; joints [13.302, 56.38, 8.114, -143.95, 68.907, 165.321]
  Set speed (17.1 mm/s)
  Call Extruder(1394.72824)
  MoveL 6129 to (456.62, 546.37, 108) mm, rotated rx 180 ry 0 rz 160 deg; joints [13.217, 56.232, 8.434, -144.078, 69.025, 165.461]
  Call Extruder(1399.02238)
  MoveL 6130 to (455.68, 545.47, 108) mm, rotated rx -180 ry 0 rz 160 deg; joints [13.126, 56.085, 8.754, -144.211, 69.141, 165.603]
  Call Extruder(1403.37154)
  MoveL 6131 to (454.74, 544.54, 108) mm, rotated rx 180 ry 0 rz 160 deg; joints [13.03, 55.938, 9.073, -144.348, 69.257, 165.746]
  Set speed (17.1 mm/s)
  Call Extruder(1406.70073)
  MoveL 6132 to (454.04, 543.82, 108) mm, rotated rx 180 ry 0 rz 160 deg; joints [12.955, 55.827, 9.314, -144.454, 69.345, 165.854]
  Call Extruder(1411.96082)
  MoveL 6133 to (452.96, 542.65, 108) mm, rotated rx -180 ry 0 rz 160 deg; joints [12.831, 55.656, 9.687, -144.627, 69.478, 166.024]
  Set speed (17.1 mm/s)
  Call Extruder(1415.35189)
  MoveL 6134 to (452.27, 541.89, 108) mm, rotated rx 180 ry 0 rz 160 deg; joints [12.748, 55.547, 9.923, -144.74, 69.563, 166.133]
  Set speed (17.1 mm/s)
  Call Extruder(1421.00833)
  MoveL 6135 to (451.16, 540.59, 108) mm, rotated rx 180 ry 0 rz 160 deg; joints [12.605, 55.37, 10.308, -144.933, 69.699, 166.313]
  Set speed (17.1 mm/s)
  Call Extruder(1424.81947)
  MoveL 6136 to (450.44, 539.7, 108) mm, rotated rx 180 ry 0 rz 160 deg; joints [12.505, 55.254, 10.563, -145.066, 69.788, 166.433]
  Call Extruder(1429.14227)
  MoveL 6137 to (449.63, 538.67, 108) mm, rotated rx -180 ry 0 rz 160 deg; joints [12.389, 55.124, 10.845, -145.218, 69.887, 166.567]
  Set speed (17.1 mm/s)
  Call Extruder(1433.49415)
  MoveL 6138 to (448.84, 537.62, 108) mm, rotated rx 180 ry 0 rz 160 deg; joints [12.268, 54.996, 11.124, -145.375, 69.984, 166.702]
  Call Extruder(1437.73199)
  MoveL 6139 to (448.09, 536.57, 108) mm, rotated rx -180 ry 0 rz 160 deg; joints [12.147, 54.876, 11.389, -145.53, 70.074, 166.832]
  Set speed (17.1 mm/s)
  Call Extruder(1442.08393)
  MoveL 6140 to (447.34, 535.49, 108) mm, rotated rx -180 ry 0 rz 160 deg; joints [12.02, 54.754, 11.656, -145.691, 70.165, 166.963]
  Set speed (17.1 mm/s)
  Call Extruder(1446.30713)
  MoveL 6141 to (446.64, 534.42, 108) mm, rotated rx -180 ry 0 rz 160 deg; joints [11.893, 54.639, 11.908, -145.851, 70.25, 167.09]
  Call Extruder(1450.58006)
  MoveL 6142 to (445.95, 533.33, 108) mm, rotated rx 180 ry 0 rz 160 deg; joints [11.761, 54.525, 12.157, -146.014, 70.333, 167.217]
  Set speed (17.1 mm/s)
  Call Extruder(1454.89855)
  MoveL 6143 to (445.27, 532.21, 108) mm, rotated rx 180 ry 0 rz 160 deg; joints [11.625, 54.414, 12.401, -146.182, 70.413, 167.343]
  Set speed (17.1 mm/s)
  Call Extruder(1459.26685)
  MoveL 6144 to (444.62, 531.07, 108) mm, rotated rx 180 ry 0 rz 160 deg; joints [11.484, 54.305, 12.642, -146.354, 70.492, 167.469]
  Call Extruder(1463.42862)
  MoveL 6145 to (444.01, 529.96, 108) mm, rotated rx -180 ry 0 rz 160 deg; joints [11.346, 54.203, 12.866, -146.52, 70.564, 167.588]
  Set speed (17.1 mm/s)
  Call Extruder(1467.73988)
  MoveL 6146 to (443.41, 528.81, 108) mm, rotated rx 180 ry 0 rz 160 deg; joints [11.201, 54.101, 13.09, -146.694, 70.635, 167.71]
  Set speed (17.1 mm/s)
  Call Extruder(1471.99211)
  MoveL 6147 to (442.83, 527.65, 108) mm, rotated rx 180 ry 0 rz 160 deg; joints [11.055, 54.004, 13.305, -146.868, 70.702, 167.828]
  Set speed (17.1 mm/s)
  Call Extruder(1476.44179)
  MoveL 6148 to (442.27, 526.43, 108) mm, rotated rx 180 ry 0 rz 160 deg; joints [10.898, 53.906, 13.52, -147.053, 70.768, 167.949]
  Set speed (17.1 mm/s)
  Call Extruder(1480.72927)
  MoveL 6149 to (441.73, 525.25, 108) mm, rotated rx -180 ry 0 rz 160 deg; joints [10.746, 53.814, 13.724, -147.232, 70.83, 168.065]
  Set speed (17.1 mm/s)
  Call Extruder(1485.02174)
  MoveL 6150 to (441.24, 524.05, 108) mm, rotated rx -180 ry 0 rz 160 deg; joints [10.589, 53.727, 13.917, -147.414, 70.887, 168.179]
  Set speed (17.0 mm/s)
  Call Extruder(1489.12520)
  MoveL 6151 to (440.77, 522.9, 108) mm, rotated rx -180 ry 0 rz 160 deg; joints [10.438, 53.645, 14.098, -147.588, 70.94, 168.287]
  Set speed (17.1 mm/s)
  Call Extruder(1497.81122)
  MoveL 6152 to (439.88, 520.43, 108) mm, rotated rx 180 ry 0 rz 160 deg; joints [10.11, 53.483, 14.457, -147.965, 71.04, 168.508]
  Set speed (17.0 mm/s)
  Call Extruder(1502.20534)
  MoveL 6153 to (439.47, 519.17, 108) mm, rotated rx 180 ry 0 rz 160 deg; joints [9.94, 53.407, 14.625, -148.158, 71.085, 168.617]
  Set speed (17.0 mm/s)
  Call Extruder(1506.26433)
  MoveL 6154 to (439.1, 518, 108) mm, rotated rx 180 ry 0 rz 160 deg; joints [9.782, 53.339, 14.776, -148.337, 71.125, 168.717]
  Call Extruder(1510.80019)
  MoveL 6155 to (438.74, 516.68, 108) mm, rotated rx 180 ry 0 rz 160 deg; joints [9.601, 53.268, 14.934, -148.539, 71.163, 168.825]
  Set speed (17.0 mm/s)
  Call Extruder(1515.05234)
  MoveL 6156 to (438.4, 515.44, 108) mm, rotated rx 180 ry 0 rz 160 deg; joints [9.431, 53.204, 15.077, -148.73, 71.198, 168.925]
  Call Extruder(1519.40482)
  MoveL 6157 to (438.1, 514.16, 108) mm, rotated rx -180 ry 0 rz 160 deg; joints [9.254, 53.143, 15.213, -148.927, 71.228, 169.025]
  Set speed (17.0 mm/s)
  Call Extruder(1523.67720)
  MoveL 6158 to (437.82, 512.9, 108) mm, rotated rx 180 ry 0 rz 160 deg; joints [9.079, 53.085, 15.341, -149.121, 71.255, 169.122]
  Set speed (17.1 mm/s)
  Call Extruder(1532.32771)
  MoveL 6159 to (437.34, 510.33, 108) mm, rotated rx 180 ry 0 rz 160 deg; joints [8.718, 52.98, 15.575, -149.517, 71.298, 169.312]
  Set speed (17.1 mm/s)
  Call Extruder(1540.90541)
  MoveL 6160 to (436.97, 507.76, 108) mm, rotated rx -180 ry 0 rz 160 deg; joints [8.353, 52.89, 15.775, -149.914, 71.326, 169.491]
  Set speed (17.1 mm/s)
  Call Extruder(1549.49162)
  MoveL 6161 to (436.71, 505.18, 108) mm, rotated rx -180 ry 0 rz 160 deg; joints [7.983, 52.815, 15.943, -150.314, 71.34, 169.663]
  Set speed (17.1 mm/s)
  Call Extruder(1557.90238)
  MoveL 6162 to (436.55, 502.63, 108) mm, rotated rx -180 ry 0 rz 160 deg; joints [7.616, 52.755, 16.076, -150.707, 71.339, 169.823]
  Call Extruder(1566.58649)
  MoveL 6163 to (436.5, 500.01, 108) mm, rotated rx 180 ry 0 rz 160 deg; joints [7.234, 52.708, 16.181, -151.115, 71.322, 169.98]
  Call Extruder(1574.38762)
  MoveL 6164 to (436.54, 497.65, 108) mm, rotated rx 180 ry 0 rz 160 deg; joints [6.888, 52.679, 16.247, -151.48, 71.294, 170.114]
  Call Extruder(0.00000)
  Call Extruder(7.63273)
  MoveL 6165 to (436.67, 495.34, 108) mm, rotated rx -180 ry 0 rz 160 deg; joints [6.548, 52.661, 16.285, -151.837, 71.255, 170.238]
  Set speed (17.1 mm/s)
  Call Extruder(15.35748)
  MoveL 6166 to (436.88, 493.01, 108) mm, rotated rx 180 ry 0 rz 160 deg; joints [6.203, 52.656, 16.298, -152.197, 71.203, 170.357]
  Set speed (17.1 mm/s)
  Call Extruder(23.06817)
  MoveL 6167 to (437.18, 490.7, 108) mm, rotated rx -180 ry 0 rz 160 deg; joints [5.859, 52.662, 16.283, -152.555, 71.138, 170.469]
  Set speed (17.1 mm/s)
  Call Extruder(30.89421)
  MoveL 6168 to (437.57, 488.36, 108) mm, rotated rx -180 ry 0 rz 160 deg; joints [5.51, 52.682, 16.241, -152.914, 71.06, 170.575]
  Set speed (17.1 mm/s)
  Call Extruder(38.52437)
  MoveL 6169 to (438.04, 486.1, 108) mm, rotated rx -180 ry 0 rz 160 deg; joints [5.172, 52.711, 16.174, -153.261, 70.972, 170.672]
  Call Extruder(46.24471)
  MoveL 6170 to (438.59, 483.83, 108) mm, rotated rx -180 ry 0 rz 160 deg; joints [4.832, 52.754, 16.079, -153.609, 70.871, 170.764]
  Call Extruder(53.87239)
  MoveL 6171 to (439.22, 481.61, 108) mm, rotated rx -180 ry 0 rz 160 deg; joints [4.499, 52.807, 15.96, -153.947, 70.758, 170.848]
  Call Extruder(61.62517)
  MoveL 6172 to (439.94, 479.38, 108) mm, rotated rx 180 ry 0 rz 160 deg; joints [4.164, 52.873, 15.814, -154.285, 70.633, 170.926]
  Call Extruder(69.46952)
  MoveL 6173 to (440.75, 477.15, 108) mm, rotated rx -180 ry 0 rz 160 deg; joints [3.829, 52.952, 15.638, -154.621, 70.492, 170.998]
  Set speed (17.1 mm/s)
  Call Extruder(76.33573)
  MoveL 6174 to (441.53, 475.22, 108) mm, rotated rx 180 ry 0 rz 160 deg; joints [3.54, 53.03, 15.464, -154.909, 70.361, 171.056]
  Set speed (17.1 mm/s)
  Call Extruder(84.82332)
  MoveL 6175 to (442.58, 472.88, 108) mm, rotated rx 180 ry 0 rz 160 deg; joints [3.19, 53.14, 15.218, -155.256, 70.184, 171.12]
  Set speed (17.1 mm/s)
  Call Extruder(92.72211)
  MoveL 6176 to (443.64, 470.74, 108) mm, rotated rx -180 ry 0 rz 160 deg; joints [2.87, 53.254, 14.964, -155.571, 70.007, 171.172]
  Call Extruder(100.35877)
  MoveL 6177 to (444.74, 468.71, 108) mm, rotated rx -180 ry 0 rz 160 deg; joints [2.567, 53.376, 14.694, -155.867, 69.826, 171.217]
  Set speed (17.1 mm/s)
  Call Extruder(108.17339)
  MoveL 6178 to (445.94, 466.68, 108) mm, rotated rx -180 ry 0 rz 160 deg; joints [2.265, 53.512, 14.392, -156.161, 69.628, 171.255]
  Set speed (17.1 mm/s)
  Call Extruder(115.81304)
  MoveL 6179 to (447.19, 464.73, 108) mm, rotated rx 180 ry 0 rz 160 deg; joints [1.978, 53.656, 14.073, -156.438, 69.424, 171.286]
  Set speed (17.1 mm/s)
  Call Extruder(123.54268)
  MoveL 6180 to (448.53, 462.81, 108) mm, rotated rx -180 ry 0 rz 160 deg; joints [1.695, 53.813, 13.727, -156.708, 69.207, 171.311]
  Set speed (17.1 mm/s)
  Call Extruder(131.35888)
  MoveL 6181 to (449.95, 460.92, 108) mm, rotated rx 180 ry 0 rz 160 deg; joints [1.417, 53.982, 13.353, -156.971, 68.978, 171.33]
  Set speed (17.1 mm/s)
  Call Extruder(138.91992)
  MoveL 6182 to (451.39, 459.14, 108) mm, rotated rx -180 ry 0 rz 160 deg; joints [1.158, 54.156, 12.97, -157.214, 68.746, 171.342]
  Set speed (17.1 mm/s)
  Call Extruder(146.72103)
  MoveL 6183 to (452.94, 457.36, 108) mm, rotated rx 180 ry 0 rz 160 deg; joints [0.9, 54.346, 12.552, -157.454, 68.496, 171.347]
  Set speed (17.1 mm/s)
  Call Extruder(154.68471)
  MoveL 6184 to (454.59, 455.61, 108) mm, rotated rx 180 ry 0 rz 160 deg; joints [0.648, 54.55, 12.103, -157.685, 68.232, 171.346]
  Call Extruder(162.14925)
  MoveL 6185 to (456.2, 454.02, 108) mm, rotated rx 180 ry 0 rz 160 deg; joints [0.421, 54.751, 11.662, -157.89, 67.976, 171.338]
  Set speed (17.1 mm/s)
  Call Extruder(169.89037)
  MoveL 6186 to (457.93, 452.44, 108) mm, rotated rx 180 ry 0 rz 160 deg; joints [0.196, 54.969, 11.184, -158.09, 67.701, 171.323]
  Set speed (17.1 mm/s)
  Call Extruder(177.70120)
  MoveL 6187 to (459.73, 450.9, 108) mm, rotated rx 180 ry 0 rz 160 deg; joints [-0.019, 55.199, 10.681, -158.279, 67.416, 171.302]
  Set speed (17.1 mm/s)
  Call Extruder(185.62069)
  MoveL 6188 to (461.6, 449.42, 108) mm, rotated rx -180 ry 0 rz 160 deg; joints [-0.226, 55.442, 10.152, -158.457, 67.118, 171.273]
  Set speed (17.1 mm/s)
  Call Extruder(193.16960)
  MoveL 6189 to (463.45, 448.07, 108) mm, rotated rx -180 ry 0 rz 160 deg; joints [-0.412, 55.682, 9.629, -158.612, 66.827, 171.239]
  Set speed (17.1 mm/s)
  Call Extruder(200.78674)
  MoveL 6190 to (465.36, 446.78, 108) mm, rotated rx 180 ry 0 rz 160 deg; joints [-0.589, 55.932, 9.085, -158.756, 66.526, 171.197]
  Set speed (17.1 mm/s)
  Call Extruder(208.61225)
  MoveL 6191 to (467.37, 445.53, 108) mm, rotated rx 180 ry 0 rz 160 deg; joints [-0.758, 56.199, 8.508, -158.89, 66.21, 171.148]
  Set speed (17.1 mm/s)
  Call Extruder(216.33344)
  MoveL 6192 to (469.39, 444.36, 108) mm, rotated rx 180 ry 0 rz 160 deg; joints [-0.914, 56.469, 7.922, -159.008, 65.891, 171.093]
  Set speed (17.1 mm/s)
  Call Extruder(224.06387)
  MoveL 6193 to (471.46, 443.27, 108) mm, rotated rx -180 ry 0 rz 160 deg; joints [-1.058, 56.748, 7.319, -159.112, 65.567, 171.03]
  Call Extruder(231.70782)
  MoveL 6194 to (473.55, 442.27, 108) mm, rotated rx 180 ry 0 rz 160 deg; joints [-1.188, 57.032, 6.708, -159.2, 65.24, 170.961]
  Call Extruder(239.51968)
  MoveL 6195 to (475.71, 441.33, 108) mm, rotated rx -180 ry 0 rz 160 deg; joints [-1.31, 57.329, 6.069, -159.276, 64.901, 170.883]
  Call Extruder(247.05493)
  MoveL 6196 to (477.83, 440.49, 108) mm, rotated rx 180 ry 0 rz 160 deg; joints [-1.415, 57.622, 5.439, -159.335, 64.57, 170.8]
  Set speed (17.1 mm/s)
  Call Extruder(254.96802)
  MoveL 6197 to (480.09, 439.7, 108) mm, rotated rx 180 ry 0 rz 160 deg; joints [-1.513, 57.937, 4.764, -159.382, 64.217, 170.706]
  Set speed (17.1 mm/s)
  Call Extruder(262.66594)
  MoveL 6198 to (482.32, 439.01, 108) mm, rotated rx 180 ry 0 rz 160 deg; joints [-1.597, 58.25, 4.096, -159.413, 63.871, 170.607]
  Set speed (17.1 mm/s)
  Call Extruder(270.33039)
  MoveL 6199 to (484.56, 438.4, 108) mm, rotated rx -180 ry 0 rz 160 deg; joints [-1.669, 58.567, 3.419, -159.429, 63.522, 170.501]
  Set speed (17.1 mm/s)
  Call Extruder(277.89312)
  MoveL 6200 to (486.79, 437.89, 108) mm, rotated rx -180 ry 0 rz 160 deg; joints [-1.728, 58.886, 2.74, -159.431, 63.176, 170.389]
  Set speed (17.1 mm/s)
  Call Extruder(285.71692)
  MoveL 6201 to (489.11, 437.44, 108) mm, rotated rx -180 ry 0 rz 160 deg; joints [-1.777, 59.221, 2.028, -159.418, 62.814, 170.265]
  Set speed (17.1 mm/s)
  Call Extruder(293.54218)
  MoveL 6202 to (491.45, 437.08, 108) mm, rotated rx -180 ry 0 rz 160 deg; joints [-1.815, 59.561, 1.306, -159.391, 62.451, 170.133]
  Call Extruder(301.32360)
  MoveL 6203 to (493.79, 436.8, 108) mm, rotated rx -180 ry 0 rz 160 deg; joints [-1.841, 59.905, 0.58, -159.348, 62.088, 169.994]
  Call Extruder(308.88157)
  MoveL 6204 to (496.07, 436.62, 108) mm, rotated rx 180 ry 0 rz 160 deg; joints [-1.855, 60.242, -0.133, -159.293, 61.734, 169.851]
  Set speed (17.1 mm/s)
  Call Extruder(316.77169)
  MoveL 6205 to (498.46, 436.52, 108) mm, rotated rx 180 ry 0 rz 160 deg; joints [-1.858, 60.599, -0.884, -159.221, 61.364, 169.694]
  Call Extruder(324.42334)
  MoveL 6206 to (500.77, 436.5, 108) mm, rotated rx 180 ry 0 rz 160 deg; joints [-1.85, 60.948, -1.619, -159.137, 61.006, 169.533]
  Call Extruder(332.21724)
  MoveL 6207 to (503.13, 436.58, 108) mm, rotated rx 180 ry 0 rz 160 deg; joints [-1.832, 61.307, -2.372, -159.037, 60.64, 169.362]
  Set speed (17.1 mm/s)
  Call Extruder(339.87329)
  MoveL 6208 to (505.44, 436.73, 108) mm, rotated rx 180 ry 0 rz 160 deg; joints [-1.803, 61.662, -3.117, -158.925, 60.282, 169.185]
  Set speed (17.1 mm/s)
  Call Extruder(347.66788)
  MoveL 6209 to (507.79, 436.98, 108) mm, rotated rx -180 ry 0 rz 160 deg; joints [-1.763, 62.026, -3.878, -158.798, 59.919, 168.997]
  Set speed (17.1 mm/s)
  Call Extruder(355.23839)
  MoveL 6210 to (510.06, 437.3, 108) mm, rotated rx -180 ry 0 rz 160 deg; joints [-1.713, 62.381, -4.62, -158.66, 59.569, 168.807]
  Call Extruder(362.87754)
  MoveL 6211 to (512.33, 437.71, 108) mm, rotated rx 180 ry 0 rz 160 deg; joints [-1.655, 62.741, -5.37, -158.509, 59.217, 168.607]
  Call Extruder(370.77930)
  MoveL 6212 to (514.67, 438.22, 108) mm, rotated rx 180 ry 0 rz 160 deg; joints [-1.584, 63.115, -6.147, -158.339, 58.856, 168.392]
  Set speed (17.1 mm/s)
  Call Extruder(378.41615)
  MoveL 6213 to (516.9, 438.79, 108) mm, rotated rx -180 ry 0 rz 160 deg; joints [-1.505, 63.476, -6.898, -158.161, 58.51, 168.177]
  Call Extruder(386.19953)
  MoveL 6214 to (519.16, 439.46, 108) mm, rotated rx 180 ry 0 rz 160 deg; joints [-1.416, 63.845, -7.662, -157.968, 58.162, 167.949]
  Set speed (17.1 mm/s)
  Call Extruder(393.81678)
  MoveL 6215 to (521.35, 440.2, 108) mm, rotated rx -180 ry 0 rz 160 deg; joints [-1.32, 64.206, -8.409, -157.766, 57.824, 167.719]
  Set speed (17.1 mm/s)
  Call Extruder(401.64711)
  MoveL 6216 to (523.57, 441.03, 108) mm, rotated rx 180 ry 0 rz 160 deg; joints [-1.213, 64.576, -9.174, -157.546, 57.482, 167.475]
  Set speed (17.1 mm/s)
  Call Extruder(409.31472)
  MoveL 6217 to (525.7, 441.94, 108) mm, rotated rx -180 ry 0 rz 160 deg; joints [-1.098, 64.937, -9.919, -157.319, 57.153, 167.228]
  Set speed (17.1 mm/s)
  Call Extruder(417.18876)
  MoveL 6218 to (527.87, 442.94, 108) mm, rotated rx 180 ry 0 rz 160 deg; joints [-0.973, 65.307, -10.679, -157.075, 56.82, 166.968]
  Call Extruder(424.72702)
  MoveL 6219 to (529.9, 443.98, 108) mm, rotated rx -180 ry 0 rz 160 deg; joints [-0.845, 65.658, -11.402, -156.83, 56.508, 166.712]
  Set speed (17.1 mm/s)
  Call Extruder(432.65025)
  MoveL 6220 to (531.99, 445.15, 108) mm, rotated rx 180 ry 0 rz 160 deg; joints [-0.702, 66.024, -12.154, -156.562, 56.187, 166.436]
  Set speed (17.1 mm/s)
  Call Extruder(440.27892)
  MoveL 6221 to (533.96, 446.34, 108) mm, rotated rx -180 ry 0 rz 160 deg; joints [-0.557, 66.374, -12.872, -156.293, 55.884, 166.164]
  Set speed (17.1 mm/s)
  Call Extruder(447.94437)
  MoveL 6222 to (535.9, 447.62, 108) mm, rotated rx -180 ry 0 rz 160 deg; joints [-0.404, 66.722, -13.583, -156.013, 55.588, 165.885]
  Set speed (17.1 mm/s)
  Call Extruder(455.72969)
  MoveL 6223 to (537.82, 448.99, 108) mm, rotated rx -180 ry 0 rz 160 deg; joints [-0.242, 67.071, -14.297, -155.72, 55.296, 165.596]
  Call Extruder(463.49743)
  MoveL 6224 to (539.68, 450.42, 108) mm, rotated rx -180 ry 0 rz 160 deg; joints [-0.073, 67.414, -14.997, -155.417, 55.013, 165.302]
  Set speed (17.1 mm/s)
  Call Extruder(471.23352)
  MoveL 6225 to (541.48, 451.92, 108) mm, rotated rx 180 ry 0 rz 160 deg; joints [0.102, 67.751, -15.684, -155.108, 54.74, 165.004]
  Call Extruder(479.00719)
  MoveL 6226 to (543.23, 453.49, 108) mm, rotated rx 180 ry 0 rz 160 deg; joints [0.284, 68.083, -16.36, -154.788, 54.476, 164.7]
  Call Extruder(486.68657)
  MoveL 6227 to (544.9, 455.1, 108) mm, rotated rx -180 ry 0 rz 160 deg; joints [0.47, 68.405, -17.016, -154.465, 54.224, 164.396]
  Set speed (17.1 mm/s)
  Call Extruder(490.91519)
  MoveL 6228 to (545.8, 456.01, 108) mm, rotated rx -180 ry 0 rz 160 deg; joints [0.575, 68.58, -17.37, -154.284, 54.09, 164.227]
  Set speed (17.1 mm/s)
  Call Extruder(495.15813)
  MoveL 6229 to (546.68, 456.95, 108) mm, rotated rx 180 ry 0 rz 160 deg; joints [0.682, 68.752, -17.72, -154.101, 53.959, 164.056]
  Set speed (17.1 mm/s)
  Call Extruder(499.49182)
  MoveL 6230 to (547.56, 457.92, 108) mm, rotated rx -180 ry 0 rz 160 deg; joints [0.793, 68.926, -18.074, -153.912, 53.829, 163.881]
  Set speed (17.1 mm/s)
  Call Extruder(503.84790)
  MoveL 6231 to (548.42, 458.92, 108) mm, rotated rx 180 ry 0 rz 160 deg; joints [0.907, 69.099, -18.424, -153.719, 53.701, 163.705]
  Set speed (17.1 mm/s)
  Call Extruder(508.12603)
  MoveL 6232 to (549.25, 459.91, 108) mm, rotated rx 180 ry 0 rz 160 deg; joints [1.019, 69.265, -18.761, -153.529, 53.58, 163.531]
  Set speed (17.1 mm/s)
  Call Extruder(512.36350)
  MoveL 6233 to (550.05, 460.92, 108) mm, rotated rx 180 ry 0 rz 160 deg; joints [1.133, 69.428, -19.091, -153.339, 53.463, 163.358]
  Set speed (17.1 mm/s)
  Call Extruder(516.60007)
  MoveL 6234 to (550.83, 461.93, 108) mm, rotated rx 180 ry 0 rz 160 deg; joints [1.247, 69.588, -19.415, -153.147, 53.35, 163.184]
  Set speed (17.1 mm/s)
  Call Extruder(521.01633)
  MoveL 6235 to (551.62, 463.01, 108) mm, rotated rx 180 ry 0 rz 160 deg; joints [1.369, 69.752, -19.746, -152.946, 53.236, 163.003]
  Set speed (17.1 mm/s)
  Call Extruder(525.39258)
  MoveL 6236 to (552.38, 464.1, 108) mm, rotated rx 180 ry 0 rz 160 deg; joints [1.49, 69.911, -20.068, -152.745, 53.127, 162.823]
  Set speed (17.1 mm/s)
  Call Extruder(529.51002)
  MoveL 6237 to (553.07, 465.13, 108) mm, rotated rx 180 ry 0 rz 160 deg; joints [1.606, 70.058, -20.364, -152.555, 53.028, 162.654]
  Set speed (17.1 mm/s)
  Call Extruder(533.74613)
  MoveL 6238 to (553.76, 466.21, 108) mm, rotated rx -180 ry 0 rz 160 deg; joints [1.727, 70.206, -20.663, -152.358, 52.93, 162.48]
  Call Extruder(538.14812)
  MoveL 6239 to (554.46, 467.34, 108) mm, rotated rx -180 ry 0 rz 160 deg; joints [1.853, 70.356, -20.967, -152.153, 52.833, 162.299]
  Call Extruder(542.35105)
  MoveL 6240 to (555.1, 468.44, 108) mm, rotated rx 180 ry 0 rz 160 deg; joints [1.975, 70.497, -21.251, -151.956, 52.744, 162.126]
